   DATA[1675,3] := 1.0;
   DATA[1675,4] := 262.657;
   DATA[1675,5] := 8.46533;
   DATA[1675,6] := 319.4053;
   DATA[1675,8] := 1.0;
   DATA[1675,9] := 1.0;
   DATA[1675,10] := 1.0;
   DATA[1675,11] := 19.71957;
   DATA[1675,12] := 2.210037;
   DATA[1675,13] := 865.9639;
   DATA[1675,14] := 1.0;
   DATA[1675,15] := 2.0;
   DATA[1675,16] := 1.0;
   DATA[1675,17] := 1.0;
   DATA[1675,18] := 1.0;
   DATA[1675,19] := 2.0;
   DATA[1675,20] := 148.808;
   DATA[1675,21] := 153.9862;
   DATA[1675,22] := 1.713261;
   DATA[1675,23] := 801.756;
   DATA[1675,24] := 2.0;
   DATA[1675,25] := 2.0;
   DATA[1675,26] := 7.876058;
   DATA[1675,27] := 142.9377;
   DATA[1675,28] := 262.6891;
   DATA[1675,29] := 12.11228;
   DATA[1675,30] := 1.721866;
   DATA[1675,31] := 1.28372;
   DATA[1675,32] := 0.7355248;
   DATA[1675,33] := 0.3082983;
   DATA[1675,34] := 2.0;
   DATA[1675,35] := 249.7597;
   DATA[1675,36] := 1.585878;
   DATA[1675,37] := 188.7016;
   DATA[1675,38] := 0.000128152;
   DATA[1675,39] := 1.0;
   DATA[1676,1] := 815.3583;
   DATA[1676,2] := 1.0;
   DATA[1676,3] := 1.0;
   DATA[1676,4] := 262.657;
   DATA[1676,5] := 8.46533;
   DATA[1676,6] := 319.5334;
   DATA[1676,8] := 1.0;
   DATA[1676,9] := 1.0;
   DATA[1676,10] := 1.0;
   DATA[1676,11] := 19.71957;
   DATA[1676,12] := 2.210037;
   DATA[1676,13] := 865.323;
   DATA[1676,14] := 1.0;
   DATA[1676,15] := 2.0;
   DATA[1676,16] := 1.0;
   DATA[1676,17] := 1.0;
   DATA[1676,18] := 1.0;
   DATA[1676,19] := 2.0;
   DATA[1676,20] := 148.808;
   DATA[1676,21] := 153.9862;
   DATA[1676,22] := 1.713261;
   DATA[1676,23] := 801.756;
   DATA[1676,24] := 2.0;
   DATA[1676,25] := 2.0;
   DATA[1676,26] := 7.876058;
   DATA[1676,27] := 142.9633;
   DATA[1676,28] := 262.6891;
   DATA[1676,29] := 12.11228;
   DATA[1676,30] := 1.721866;
   DATA[1676,31] := 1.299731;
   DATA[1676,32] := 0.7355248;
   DATA[1676,33] := 0.3084265;
   DATA[1676,34] := 2.0;
   DATA[1676,35] := 249.7597;
   DATA[1676,36] := 1.585878;
   DATA[1676,37] := 188.7016;
   DATA[1676,38] := 0.000128152;
   DATA[1676,39] := 1.0;
   DATA[1677,1] := 815.5153;
   DATA[1677,2] := 1.0;
   DATA[1677,3] := 1.0;
   DATA[1677,4] := 262.657;
   DATA[1677,5] := 8.46533;
   DATA[1677,6] := 319.5334;
   DATA[1677,8] := 1.0;
   DATA[1677,9] := 1.0;
   DATA[1677,10] := 1.0;
   DATA[1677,11] := 19.70357;
   DATA[1677,12] := 2.210037;
   DATA[1677,13] := 865.0827;
   DATA[1677,14] := 1.0;
   DATA[1677,15] := 2.0;
   DATA[1677,16] := 1.0;
   DATA[1677,17] := 1.0;
   DATA[1677,18] := 1.0;
   DATA[1677,19] := 2.0;
   DATA[1677,20] := 148.808;
   DATA[1677,21] := 154.0631;
   DATA[1677,22] := 1.713261;
   DATA[1677,23] := 801.8329;
   DATA[1677,24] := 2.0;
   DATA[1677,25] := 2.0;
   DATA[1677,26] := 7.876058;
   DATA[1677,27] := 143.1172;
   DATA[1677,28] := 262.6891;
   DATA[1677,29] := 12.11228;
   DATA[1677,30] := 1.722892;
   DATA[1677,31] := 1.301652;
   DATA[1677,32] := 0.7355248;
   DATA[1677,33] := 0.3084905;
   DATA[1677,34] := 2.0;
   DATA[1677,35] := 249.8558;
   DATA[1677,36] := 1.585878;
   DATA[1677,37] := 188.7016;
   DATA[1677,38] := 0.000128152;
   DATA[1677,39] := 1.0;
   DATA[1678,1] := 815.5938;
   DATA[1678,2] := 1.0;
   DATA[1678,3] := 1.0;
   DATA[1678,4] := 262.657;
   DATA[1678,5] := 8.46533;
   DATA[1678,6] := 319.5334;
   DATA[1678,8] := 1.0;
   DATA[1678,9] := 1.0;
   DATA[1678,10] := 1.0;
   DATA[1678,11] := 19.68436;
   DATA[1678,12] := 2.210037;
   DATA[1678,13] := 864.4819;
   DATA[1678,14] := 1.0;
   DATA[1678,15] := 2.0;
   DATA[1678,16] := 1.0;
   DATA[1678,17] := 1.0;
   DATA[1678,18] := 1.0;
   DATA[1678,19] := 2.0;
   DATA[1678,20] := 148.808;
   DATA[1678,21] := 154.1912;
   DATA[1678,22] := 1.711082;
   DATA[1678,23] := 802.2174;
   DATA[1678,24] := 2.0;
   DATA[1678,25] := 2.0;
   DATA[1678,26] := 7.876058;
   DATA[1678,27] := 143.1172;
   DATA[1678,28] := 262.6891;
   DATA[1678,29] := 12.11228;
   DATA[1678,30] := 1.723789;
   DATA[1678,31] := 1.301652;
   DATA[1678,32] := 0.7355248;
   DATA[1678,33] := 0.3084905;
   DATA[1678,34] := 2.0;
   DATA[1678,35] := 249.9359;
   DATA[1678,36] := 1.585878;
   DATA[1678,37] := 188.7016;
   DATA[1678,38] := 0.000128152;
   DATA[1678,39] := 1.0;
   DATA[1679,1] := 815.4761;
   DATA[1679,2] := 1.0;
   DATA[1679,3] := 1.0;
   DATA[1679,4] := 262.657;
   DATA[1679,5] := 8.46533;
   DATA[1679,6] := 319.5334;
   DATA[1679,8] := 1.0;
   DATA[1679,9] := 1.0;
   DATA[1679,10] := 1.0;
   DATA[1679,11] := 19.68436;
   DATA[1679,12] := 2.210037;
   DATA[1679,13] := 864.2816;
   DATA[1679,14] := 1.0;
   DATA[1679,15] := 2.0;
   DATA[1679,16] := 1.0;
   DATA[1679,17] := 1.0;
   DATA[1679,18] := 1.0;
   DATA[1679,19] := 2.0;
   DATA[1679,20] := 148.808;
   DATA[1679,21] := 154.1912;
   DATA[1679,22] := 1.711082;
   DATA[1679,23] := 802.4097;
   DATA[1679,24] := 2.0;
   DATA[1679,25] := 2.0;
   DATA[1679,26] := 7.876058;
   DATA[1679,27] := 143.1172;
   DATA[1679,28] := 262.6891;
   DATA[1679,29] := 12.11228;
   DATA[1679,30] := 1.723789;
   DATA[1679,31] := 1.289484;
   DATA[1679,32] := 0.7355248;
   DATA[1679,33] := 0.3084905;
   DATA[1679,34] := 2.0;
   DATA[1679,35] := 249.9359;
   DATA[1679,36] := 1.585878;
   DATA[1679,37] := 188.7337;
   DATA[1679,38] := 0.000128152;
   DATA[1679,39] := 1.0;
   DATA[1680,1] := 815.3583;
   DATA[1680,2] := 1.0;
   DATA[1680,3] := 1.0;
   DATA[1680,4] := 262.657;
   DATA[1680,5] := 8.46533;
   DATA[1680,6] := 319.5334;
   DATA[1680,8] := 1.0;
   DATA[1680,9] := 1.0;
   DATA[1680,10] := 1.0;
   DATA[1680,11] := 19.68436;
   DATA[1680,12] := 2.210037;
   DATA[1680,13] := 863.7209;
   DATA[1680,14] := 1.0;
   DATA[1680,15] := 2.0;
   DATA[1680,16] := 1.0;
   DATA[1680,17] := 1.0;
   DATA[1680,18] := 1.0;
   DATA[1680,19] := 2.0;
   DATA[1680,20] := 148.808;
   DATA[1680,21] := 154.1912;
   DATA[1680,22] := 1.711082;
   DATA[1680,23] := 802.4866;
   DATA[1680,24] := 2.0;
   DATA[1680,25] := 2.0;
   DATA[1680,26] := 7.876058;
   DATA[1680,27] := 143.1172;
   DATA[1680,28] := 262.6891;
   DATA[1680,29] := 12.11228;
   DATA[1680,30] := 1.723789;
   DATA[1680,31] := 1.275522;
   DATA[1680,32] := 0.7355248;
   DATA[1680,33] := 0.3084905;
   DATA[1680,34] := 2.0;
   DATA[1680,35] := 249.9359;
   DATA[1680,36] := 1.601897;
   DATA[1680,37] := 188.8138;
   DATA[1680,38] := 0.000128152;
   DATA[1680,39] := 1.0;
   DATA[1681,1] := 815.319;
   DATA[1681,2] := 1.0;
   DATA[1681,3] := 1.0;
   DATA[1681,4] := 262.657;
   DATA[1681,5] := 8.46533;
   DATA[1681,6] := 319.5334;
   DATA[1681,8] := 1.0;
   DATA[1681,9] := 1.0;
   DATA[1681,10] := 1.0;
   DATA[1681,11] := 19.73238;
   DATA[1681,12] := 2.210037;
   DATA[1681,13] := 863.2402;
   DATA[1681,14] := 1.0;
   DATA[1681,15] := 2.0;
   DATA[1681,16] := 1.0;
   DATA[1681,17] := 1.0;
   DATA[1681,18] := 1.0;
   DATA[1681,19] := 2.0;
   DATA[1681,20] := 148.808;
   DATA[1681,21] := 154.1912;
   DATA[1681,22] := 1.711979;
   DATA[1681,23] := 802.871;
   DATA[1681,24] := 2.0;
   DATA[1681,25] := 2.0;
   DATA[1681,26] := 7.876058;
   DATA[1681,27] := 143.1172;
   DATA[1681,28] := 262.6891;
   DATA[1681,29] := 12.11228;
   DATA[1681,30] := 1.725327;
   DATA[1681,31] := 1.277315;
   DATA[1681,32] := 0.7355248;
   DATA[1681,33] := 0.3084905;
   DATA[1681,34] := 2.0;
   DATA[1681,35] := 249.9359;
   DATA[1681,36] := 1.681991;
   DATA[1681,37] := 188.8458;
   DATA[1681,38] := 0.000128152;
   DATA[1681,39] := 1.0;
   DATA[1682,1] := 815.319;
   DATA[1682,2] := 1.0;
   DATA[1682,3] := 1.0;
   DATA[1682,4] := 262.657;
   DATA[1682,5] := 8.46533;
   DATA[1682,6] := 319.5334;
   DATA[1682,8] := 1.0;
   DATA[1682,9] := 1.0;
   DATA[1682,10] := 1.0;
   DATA[1682,11] := 19.7868;
   DATA[1682,12] := 2.209397;
   DATA[1682,13] := 863.2803;
   DATA[1682,14] := 1.0;
   DATA[1682,15] := 2.0;
   DATA[1682,16] := 1.0;
   DATA[1682,17] := 1.0;
   DATA[1682,18] := 1.0;
   DATA[1682,19] := 2.0;
   DATA[1682,20] := 148.808;
   DATA[1682,21] := 154.1912;
   DATA[1682,22] := 1.712748;
   DATA[1682,23] := 803.4094;
   DATA[1682,24] := 2.0;
   DATA[1682,25] := 2.0;
   DATA[1682,26] := 7.876058;
   DATA[1682,27] := 143.0659;
   DATA[1682,28] := 262.6891;
   DATA[1682,29] := 12.11228;
   DATA[1682,30] := 1.725327;
   DATA[1682,31] := 1.276547;
   DATA[1682,32] := 0.7355248;
   DATA[1682,33] := 0.3084905;
   DATA[1682,34] := 2.0;
   DATA[1682,35] := 249.9359;
   DATA[1682,36] := 1.681991;
   DATA[1682,37] := 188.8458;
   DATA[1682,38] := 0.000128152;
   DATA[1682,39] := 1.0;
   DATA[1683,1] := 815.3975;
   DATA[1683,2] := 1.0;
   DATA[1683,3] := 1.0;
   DATA[1683,4] := 262.657;
   DATA[1683,5] := 8.46533;
   DATA[1683,6] := 319.5334;
   DATA[1683,8] := 1.0;
   DATA[1683,9] := 1.0;
   DATA[1683,10] := 1.0;
   DATA[1683,11] := 19.7868;
   DATA[1683,12] := 2.209397;
   DATA[1683,13] := 862.5593;
   DATA[1683,14] := 1.0;
   DATA[1683,15] := 2.0;
   DATA[1683,16] := 1.0;
   DATA[1683,17] := 1.0;
   DATA[1683,18] := 1.0;
   DATA[1683,19] := 2.0;
   DATA[1683,20] := 148.808;
   DATA[1683,21] := 154.1912;
   DATA[1683,22] := 1.712748;
   DATA[1683,23] := 803.4094;
   DATA[1683,24] := 2.0;
   DATA[1683,25] := 2.0;
   DATA[1683,26] := 7.876058;
   DATA[1683,27] := 143.0659;
   DATA[1683,28] := 262.6891;
   DATA[1683,29] := 12.11228;
   DATA[1683,30] := 1.725327;
   DATA[1683,31] := 1.27834;
   DATA[1683,32] := 0.7355248;
   DATA[1683,33] := 0.3084905;
   DATA[1683,34] := 2.0;
   DATA[1683,35] := 249.9359;
   DATA[1683,36] := 1.681991;
   DATA[1683,37] := 188.8458;
   DATA[1683,38] := 0.000128152;
   DATA[1683,39] := 1.0;
   DATA[1684,1] := 815.1228;
   DATA[1684,2] := 1.0;
   DATA[1684,3] := 1.0;
   DATA[1684,4] := 262.657;
   DATA[1684,5] := 8.46533;
   DATA[1684,6] := 319.5334;
   DATA[1684,8] := 1.0;
   DATA[1684,9] := 1.0;
   DATA[1684,10] := 1.0;
   DATA[1684,11] := 19.72277;
   DATA[1684,12] := 2.209397;
   DATA[1684,13] := 862.4391;
   DATA[1684,14] := 1.0;
   DATA[1684,15] := 2.0;
   DATA[1684,16] := 1.0;
   DATA[1684,17] := 1.0;
   DATA[1684,18] := 1.0;
   DATA[1684,19] := 2.0;
   DATA[1684,20] := 148.808;
   DATA[1684,21] := 154.1912;
   DATA[1684,22] := 1.712748;
   DATA[1684,23] := 803.8323;
   DATA[1684,24] := 2.0;
   DATA[1684,25] := 2.0;
   DATA[1684,26] := 7.876058;
   DATA[1684,27] := 143.0659;
   DATA[1684,28] := 262.6891;
   DATA[1684,29] := 12.11228;
   DATA[1684,30] := 1.725327;
   DATA[1684,31] := 1.272064;
   DATA[1684,32] := 0.7355248;
   DATA[1684,33] := 0.3084905;
   DATA[1684,34] := 2.0;
   DATA[1684,35] := 249.9359;
   DATA[1684,36] := 1.665972;
   DATA[1684,37] := 188.8458;
   DATA[1684,38] := 0.000128152;
   DATA[1684,39] := 1.0;
   DATA[1685,1] := 815.0835;
   DATA[1685,2] := 1.0;
   DATA[1685,3] := 1.0;
   DATA[1685,4] := 262.657;
   DATA[1685,5] := 8.46533;
   DATA[1685,6] := 319.5334;
   DATA[1685,8] := 1.0;
   DATA[1685,9] := 1.0;
   DATA[1685,10] := 1.0;
   DATA[1685,11] := 19.70357;
   DATA[1685,12] := 2.209397;
   DATA[1685,13] := 862.0386;
   DATA[1685,14] := 1.0;
   DATA[1685,15] := 2.0;
   DATA[1685,16] := 1.0;
   DATA[1685,17] := 1.0;
   DATA[1685,18] := 1.0;
   DATA[1685,19] := 2.0;
   DATA[1685,20] := 148.808;
   DATA[1685,21] := 154.1912;
   DATA[1685,22] := 1.712876;
   DATA[1685,23] := 803.6016;
   DATA[1685,24] := 2.0;
   DATA[1685,25] := 2.0;
   DATA[1685,26] := 7.876058;
   DATA[1685,27] := 143.0659;
   DATA[1685,28] := 262.6891;
   DATA[1685,29] := 12.11228;
   DATA[1685,30] := 1.725327;
   DATA[1685,31] := 1.271935;
   DATA[1685,32] := 0.7355248;
   DATA[1685,33] := 0.3084905;
   DATA[1685,34] := 2.0;
   DATA[1685,35] := 249.9359;
   DATA[1685,36] := 1.649953;
   DATA[1685,37] := 188.8458;
   DATA[1685,38] := 0.000128152;
   DATA[1685,39] := 1.0;
   DATA[1686,1] := 815.3975;
   DATA[1686,2] := 1.0;
   DATA[1686,3] := 1.0;
   DATA[1686,4] := 262.657;
   DATA[1686,5] := 8.46533;
   DATA[1686,6] := 319.5334;
   DATA[1686,8] := 1.0;
   DATA[1686,9] := 1.0;
   DATA[1686,10] := 1.0;
   DATA[1686,11] := 19.70357;
   DATA[1686,12] := 2.209397;
   DATA[1686,13] := 861.7582;
   DATA[1686,14] := 1.0;
   DATA[1686,15] := 2.0;
   DATA[1686,16] := 1.0;
   DATA[1686,17] := 1.0;
   DATA[1686,18] := 1.0;
   DATA[1686,19] := 2.0;
   DATA[1686,20] := 148.808;
   DATA[1686,21] := 154.1912;
   DATA[1686,22] := 1.712876;
   DATA[1686,23] := 803.6016;
   DATA[1686,24] := 2.0;
   DATA[1686,25] := 2.0;
   DATA[1686,26] := 7.876058;
   DATA[1686,27] := 143.0659;
   DATA[1686,28] := 262.6891;
   DATA[1686,29] := 12.11228;
   DATA[1686,30] := 1.725327;
   DATA[1686,31] := 1.270911;
   DATA[1686,32] := 0.7355248;
   DATA[1686,33] := 0.3084905;
   DATA[1686,34] := 2.0;
   DATA[1686,35] := 249.9359;
   DATA[1686,36] := 1.649953;
   DATA[1686,37] := 188.8458;
   DATA[1686,38] := 0.000128152;
   DATA[1686,39] := 1.0;
   DATA[1687,1] := 815.2798;
   DATA[1687,2] := 1.0;
   DATA[1687,3] := 1.0;
   DATA[1687,4] := 262.657;
   DATA[1687,5] := 8.46533;
   DATA[1687,6] := 319.5334;
   DATA[1687,8] := 1.0;
   DATA[1687,9] := 1.0;
   DATA[1687,10] := 1.0;
   DATA[1687,11] := 19.76439;
   DATA[1687,12] := 2.214649;
   DATA[1687,13] := 860.9572;
   DATA[1687,14] := 1.0;
   DATA[1687,15] := 2.0;
   DATA[1687,16] := 1.0;
   DATA[1687,17] := 1.0;
   DATA[1687,18] := 1.0;
   DATA[1687,19] := 2.0;
   DATA[1687,20] := 148.808;
   DATA[1687,21] := 154.1912;
   DATA[1687,22] := 1.712876;
   DATA[1687,23] := 803.4094;
   DATA[1687,24] := 2.0;
   DATA[1687,25] := 2.0;
   DATA[1687,26] := 7.876058;
   DATA[1687,27] := 143.0659;
   DATA[1687,28] := 262.6891;
   DATA[1687,29] := 12.11228;
   DATA[1687,30] := 1.724045;
   DATA[1687,31] := 1.270398;
   DATA[1687,32] := 0.7355248;
   DATA[1687,33] := 0.3084905;
   DATA[1687,34] := 2.0;
   DATA[1687,35] := 249.9359;
   DATA[1687,36] := 1.649953;
   DATA[1687,37] := 188.8458;
   DATA[1687,38] := 0.000128152;
   DATA[1687,39] := 1.0;
   DATA[1688,1] := 815.2013;
   DATA[1688,2] := 1.0;
   DATA[1688,3] := 1.0;
   DATA[1688,4] := 262.657;
   DATA[1688,5] := 8.46533;
   DATA[1688,6] := 319.5334;
   DATA[1688,8] := 1.0;
   DATA[1688,9] := 1.0;
   DATA[1688,10] := 1.0;
   DATA[1688,11] := 19.76439;
   DATA[1688,12] := 2.214649;
   DATA[1688,13] := 860.5566;
   DATA[1688,14] := 1.0;
   DATA[1688,15] := 2.0;
   DATA[1688,16] := 1.0;
   DATA[1688,17] := 1.0;
   DATA[1688,18] := 1.0;
   DATA[1688,19] := 2.0;
   DATA[1688,20] := 148.808;
   DATA[1688,21] := 154.1912;
   DATA[1688,22] := 1.712876;
   DATA[1688,23] := 803.294;
   DATA[1688,24] := 2.0;
   DATA[1688,25] := 2.0;
   DATA[1688,26] := 7.876058;
   DATA[1688,27] := 143.0659;
   DATA[1688,28] := 262.6891;
   DATA[1688,29] := 12.11228;
   DATA[1688,30] := 1.724045;
   DATA[1688,31] := 1.287306;
   DATA[1688,32] := 0.7355248;
   DATA[1688,33] := 0.3084905;
   DATA[1688,34] := 2.0;
   DATA[1688,35] := 249.9359;
   DATA[1688,36] := 1.649953;
   DATA[1688,37] := 188.8458;
   DATA[1688,38] := 0.000128152;
   DATA[1688,39] := 1.0;
   DATA[1689,1] := 815.4761;
   DATA[1689,2] := 1.0;
   DATA[1689,3] := 1.0;
   DATA[1689,4] := 262.657;
   DATA[1689,5] := 8.46533;
   DATA[1689,6] := 319.5334;
   DATA[1689,8] := 1.0;
   DATA[1689,9] := 1.0;
   DATA[1689,10] := 1.0;
   DATA[1689,11] := 19.77399;
   DATA[1689,12] := 2.215418;
   DATA[1689,13] := 860.0359;
   DATA[1689,14] := 1.0;
   DATA[1689,15] := 2.0;
   DATA[1689,16] := 1.0;
   DATA[1689,17] := 1.0;
   DATA[1689,18] := 1.0;
   DATA[1689,19] := 2.0;
   DATA[1689,20] := 148.808;
   DATA[1689,21] := 154.1912;
   DATA[1689,22] := 1.712876;
   DATA[1689,23] := 803.4863;
   DATA[1689,24] := 2.0;
   DATA[1689,25] := 2.0;
   DATA[1689,26] := 7.876058;
   DATA[1689,27] := 143.0659;
   DATA[1689,28] := 262.6891;
   DATA[1689,29] := 12.11228;
   DATA[1689,30] := 1.722251;
   DATA[1689,31] := 1.291918;
   DATA[1689,32] := 0.7355248;
   DATA[1689,33] := 0.3084905;
   DATA[1689,34] := 2.0;
   DATA[1689,35] := 249.9359;
   DATA[1689,36] := 1.649953;
   DATA[1689,37] := 188.8458;
   DATA[1689,38] := 0.000128152;
   DATA[1689,39] := 1.0;
   DATA[1690,1] := 815.2013;
   DATA[1690,2] := 1.0;
   DATA[1690,3] := 1.0;
   DATA[1690,4] := 262.657;
   DATA[1690,5] := 8.46533;
   DATA[1690,6] := 319.5334;
   DATA[1690,8] := 1.0;
   DATA[1690,9] := 1.0;
   DATA[1690,10] := 1.0;
   DATA[1690,11] := 19.7804;
   DATA[1690,12] := 2.21593;
   DATA[1690,13] := 859.8757;
   DATA[1690,14] := 1.0;
   DATA[1690,15] := 2.0;
   DATA[1690,16] := 1.0;
   DATA[1690,17] := 1.0;
   DATA[1690,18] := 1.0;
   DATA[1690,19] := 2.0;
   DATA[1690,20] := 148.808;
   DATA[1690,21] := 154.1912;
   DATA[1690,22] := 1.712876;
   DATA[1690,23] := 803.6401;
   DATA[1690,24] := 2.0;
   DATA[1690,25] := 2.0;
   DATA[1690,26] := 7.876058;
   DATA[1690,27] := 143.0659;
   DATA[1690,28] := 262.6891;
   DATA[1690,29] := 12.11228;
   DATA[1690,30] := 1.721866;
   DATA[1690,31] := 1.291918;
   DATA[1690,32] := 0.7355248;
   DATA[1690,33] := 0.3084905;
   DATA[1690,34] := 2.0;
   DATA[1690,35] := 250.0961;
   DATA[1690,36] := 1.649953;
   DATA[1690,37] := 188.8458;
   DATA[1690,38] := 0.000128152;
   DATA[1690,39] := 1.0;
   DATA[1691,1] := 815.0835;
   DATA[1691,2] := 1.0;
   DATA[1691,3] := 1.0;
   DATA[1691,4] := 262.657;
   DATA[1691,5] := 8.46533;
   DATA[1691,6] := 319.5334;
   DATA[1691,8] := 1.0;
   DATA[1691,9] := 1.0;
   DATA[1691,10] := 1.0;
   DATA[1691,11] := 19.7804;
   DATA[1691,12] := 2.21593;
   DATA[1691,13] := 858.8743;
   DATA[1691,14] := 1.0;
   DATA[1691,15] := 2.0;
   DATA[1691,16] := 1.0;
   DATA[1691,17] := 1.0;
   DATA[1691,18] := 1.0;
   DATA[1691,19] := 2.0;
   DATA[1691,20] := 148.808;
   DATA[1691,21] := 154.1912;
   DATA[1691,22] := 1.712107;
   DATA[1691,23] := 803.8323;
   DATA[1691,24] := 2.0;
   DATA[1691,25] := 2.0;
   DATA[1691,26] := 7.876058;
   DATA[1691,27] := 143.0659;
   DATA[1691,28] := 262.6891;
   DATA[1691,29] := 12.11228;
   DATA[1691,30] := 1.721866;
   DATA[1691,31] := 1.282567;
   DATA[1691,32] := 0.7355248;
   DATA[1691,33] := 0.3084905;
   DATA[1691,34] := 2.0;
   DATA[1691,35] := 250.0961;
   DATA[1691,36] := 1.537821;
   DATA[1691,37] := 188.8458;
   DATA[1691,38] := 0.000128152;
   DATA[1691,39] := 1.0;
   DATA[1692,1] := 814.8088;
   DATA[1692,2] := 1.0;
   DATA[1692,3] := 1.0;
   DATA[1692,4] := 262.657;
   DATA[1692,5] := 8.46533;
   DATA[1692,6] := 319.5334;
   DATA[1692,8] := 1.0;
   DATA[1692,9] := 1.0;
   DATA[1692,10] := 1.0;
   DATA[1692,11] := 19.80601;
   DATA[1692,12] := 2.21593;
   DATA[1692,13] := 858.3536;
   DATA[1692,14] := 1.0;
   DATA[1692,15] := 2.0;
   DATA[1692,16] := 1.0;
   DATA[1692,17] := 1.0;
   DATA[1692,18] := 1.0;
   DATA[1692,19] := 2.0;
   DATA[1692,20] := 148.808;
   DATA[1692,21] := 154.1912;
   DATA[1692,22] := 1.710057;
   DATA[1692,23] := 804.4476;
   DATA[1692,24] := 2.0;
   DATA[1692,25] := 2.0;
   DATA[1692,26] := 7.876058;
   DATA[1692,27] := 143.0659;
   DATA[1692,28] := 262.6891;
   DATA[1692,29] := 12.11228;
   DATA[1692,30] := 1.721866;
   DATA[1692,31] := 1.281927;
   DATA[1692,32] := 0.7353967;
   DATA[1692,33] := 0.3084905;
   DATA[1692,34] := 2.0;
   DATA[1692,35] := 250.0961;
   DATA[1692,36] := 1.537821;
   DATA[1692,37] := 188.8458;
   DATA[1692,38] := 0.000128152;
   DATA[1692,39] := 1.0;
   DATA[1693,1] := 814.7302;
   DATA[1693,2] := 1.0;
   DATA[1693,3] := 1.0;
   DATA[1693,4] := 262.657;
   DATA[1693,5] := 8.46533;
   DATA[1693,6] := 319.5334;
   DATA[1693,8] := 1.0;
   DATA[1693,9] := 1.0;
   DATA[1693,10] := 1.0;
   DATA[1693,11] := 19.83802;
   DATA[1693,12] := 2.21593;
   DATA[1693,13] := 857.6327;
   DATA[1693,14] := 1.0;
   DATA[1693,15] := 2.0;
   DATA[1693,16] := 1.0;
   DATA[1693,17] := 1.0;
   DATA[1693,18] := 1.0;
   DATA[1693,19] := 2.0;
   DATA[1693,20] := 148.808;
   DATA[1693,21] := 154.1912;
   DATA[1693,22] := 1.710057;
   DATA[1693,23] := 804.7167;
   DATA[1693,24] := 2.0;
   DATA[1693,25] := 2.0;
   DATA[1693,26] := 7.876058;
   DATA[1693,27] := 143.0659;
   DATA[1693,28] := 262.6891;
   DATA[1693,29] := 12.11228;
   DATA[1693,30] := 1.721866;
   DATA[1693,31] := 1.281927;
   DATA[1693,32] := 0.7353967;
   DATA[1693,33] := 0.3084905;
   DATA[1693,34] := 2.0;
   DATA[1693,35] := 250.016;
   DATA[1693,36] := 1.569859;
   DATA[1693,37] := 188.8458;
   DATA[1693,38] := 0.000128152;
   DATA[1693,39] := 1.0;
   DATA[1694,1] := 814.7302;
   DATA[1694,2] := 1.0;
   DATA[1694,3] := 1.0;
   DATA[1694,4] := 262.657;
   DATA[1694,5] := 8.46533;
   DATA[1694,6] := 319.5334;
   DATA[1694,8] := 1.0;
   DATA[1694,9] := 1.0;
   DATA[1694,10] := 1.0;
   DATA[1694,11] := 19.83802;
   DATA[1694,12] := 2.21593;
   DATA[1694,13] := 857.6327;
   DATA[1694,14] := 1.0;
   DATA[1694,15] := 2.0;
   DATA[1694,16] := 1.0;
   DATA[1694,17] := 1.0;
   DATA[1694,18] := 1.0;
   DATA[1694,19] := 2.0;
   DATA[1694,20] := 148.808;
   DATA[1694,21] := 154.1912;
   DATA[1694,22] := 1.710057;
   DATA[1694,23] := 804.7167;
   DATA[1694,24] := 2.0;
   DATA[1694,25] := 2.0;
   DATA[1694,26] := 7.876058;
   DATA[1694,27] := 143.0659;
   DATA[1694,28] := 262.6891;
   DATA[1694,29] := 12.11228;
   DATA[1694,30] := 1.721866;
   DATA[1694,31] := 1.281927;
   DATA[1694,32] := 0.7353967;
   DATA[1694,33] := 0.3084905;
   DATA[1694,34] := 2.0;
   DATA[1694,35] := 250.016;
   DATA[1694,36] := 1.569859;
   DATA[1694,37] := 188.8458;
   DATA[1694,38] := 0.000128152;
   DATA[1694,39] := 1.0;
   DATA[1695,1] := 814.8088;
   DATA[1695,2] := 1.0;
   DATA[1695,3] := 1.0;
   DATA[1695,4] := 262.657;
   DATA[1695,5] := 8.46533;
   DATA[1695,6] := 319.5334;
   DATA[1695,8] := 1.0;
   DATA[1695,9] := 1.0;
   DATA[1695,10] := 1.0;
   DATA[1695,11] := 19.83802;
   DATA[1695,12] := 2.21593;
   DATA[1695,13] := 857.3523;
   DATA[1695,14] := 1.0;
   DATA[1695,15] := 2.0;
   DATA[1695,16] := 1.0;
   DATA[1695,17] := 1.0;
   DATA[1695,18] := 1.0;
   DATA[1695,19] := 2.0;
   DATA[1695,20] := 148.808;
   DATA[1695,21] := 154.1912;
   DATA[1695,22] := 1.710057;
   DATA[1695,23] := 804.6398;
   DATA[1695,24] := 2.0;
   DATA[1695,25] := 2.0;
   DATA[1695,26] := 7.876058;
   DATA[1695,27] := 143.2197;
   DATA[1695,28] := 262.6891;
   DATA[1695,29] := 12.11228;
   DATA[1695,30] := 1.721866;
   DATA[1695,31] := 1.290509;
   DATA[1695,32] := 0.7353967;
   DATA[1695,33] := 0.3084905;
   DATA[1695,34] := 2.0;
   DATA[1695,35] := 249.984;
   DATA[1695,36] := 1.681991;
   DATA[1695,37] := 188.8458;
   DATA[1695,38] := 0.000128152;
   DATA[1695,39] := 1.0;
   DATA[1696,1] := 814.9265;
   DATA[1696,2] := 1.0;
   DATA[1696,3] := 1.0;
   DATA[1696,4] := 262.657;
   DATA[1696,5] := 8.46533;
   DATA[1696,6] := 319.5334;
   DATA[1696,8] := 1.0;
   DATA[1696,9] := 1.0;
   DATA[1696,10] := 1.0;
   DATA[1696,11] := 19.83802;
   DATA[1696,12] := 2.21593;
   DATA[1696,13] := 856.8716;
   DATA[1696,14] := 1.0;
   DATA[1696,15] := 2.0;
   DATA[1696,16] := 1.0;
   DATA[1696,17] := 1.0;
   DATA[1696,18] := 1.0;
   DATA[1696,19] := 2.0;
   DATA[1696,20] := 148.808;
   DATA[1696,21] := 154.1912;
   DATA[1696,22] := 1.711595;
   DATA[1696,23] := 804.3707;
   DATA[1696,24] := 2.0;
   DATA[1696,25] := 2.0;
   DATA[1696,26] := 7.876058;
   DATA[1696,27] := 143.2197;
   DATA[1696,28] := 262.6891;
   DATA[1696,29] := 12.11228;
   DATA[1696,30] := 1.722892;
   DATA[1696,31] := 1.291789;
   DATA[1696,32] := 0.7353967;
   DATA[1696,33] := 0.3084905;
   DATA[1696,34] := 2.0;
   DATA[1696,35] := 249.984;
   DATA[1696,36] := 1.681991;
   DATA[1696,37] := 188.8458;
   DATA[1696,38] := 0.000128152;
   DATA[1696,39] := 1.0;
   DATA[1697,1] := 814.8088;
   DATA[1697,2] := 1.0;
   DATA[1697,3] := 1.0;
   DATA[1697,4] := 262.657;
   DATA[1697,5] := 8.46533;
   DATA[1697,6] := 319.5334;
   DATA[1697,8] := 1.0;
   DATA[1697,9] := 1.0;
   DATA[1697,10] := 1.0;
   DATA[1697,11] := 19.73878;
   DATA[1697,12] := 2.214265;
   DATA[1697,13] := 856.9117;
   DATA[1697,14] := 1.0;
   DATA[1697,15] := 2.0;
   DATA[1697,16] := 1.0;
   DATA[1697,17] := 1.0;
   DATA[1697,18] := 1.0;
   DATA[1697,19] := 2.0;
   DATA[1697,20] := 148.808;
   DATA[1697,21] := 154.1912;
   DATA[1697,22] := 1.711595;
   DATA[1697,23] := 804.0246;
   DATA[1697,24] := 2.0;
   DATA[1697,25] := 2.0;
   DATA[1697,26] := 7.876058;
   DATA[1697,27] := 143.2197;
   DATA[1697,28] := 262.625;
   DATA[1697,29] := 12.11228;
   DATA[1697,30] := 1.723661;
   DATA[1697,31] := 1.282439;
   DATA[1697,32] := 0.7353967;
   DATA[1697,33] := 0.3084905;
   DATA[1697,34] := 2.0;
   DATA[1697,35] := 249.984;
   DATA[1697,36] := 1.681991;
   DATA[1697,37] := 188.8458;
   DATA[1697,38] := 0.000128152;
   DATA[1697,39] := 1.0;
   DATA[1698,1] := 815.162;
   DATA[1698,2] := 1.0;
   DATA[1698,3] := 1.0;
   DATA[1698,4] := 262.657;
   DATA[1698,5] := 8.46533;
   DATA[1698,6] := 319.5334;
   DATA[1698,8] := 1.0;
   DATA[1698,9] := 1.0;
   DATA[1698,10] := 1.0;
   DATA[1698,11] := 19.70357;
   DATA[1698,12] := 2.214265;
   DATA[1698,13] := 856.0706;
   DATA[1698,14] := 1.0;
   DATA[1698,15] := 2.0;
   DATA[1698,16] := 1.0;
   DATA[1698,17] := 1.0;
   DATA[1698,18] := 1.0;
   DATA[1698,19] := 2.0;
   DATA[1698,20] := 148.808;
   DATA[1698,21] := 154.1912;
   DATA[1698,22] := 1.711595;
   DATA[1698,23] := 804.8321;
   DATA[1698,24] := 2.0;
   DATA[1698,25] := 2.0;
   DATA[1698,26] := 7.876058;
   DATA[1698,27] := 143.2197;
   DATA[1698,28] := 262.3366;
   DATA[1698,29] := 12.11228;
   DATA[1698,30] := 1.723661;
   DATA[1698,31] := 1.282439;
   DATA[1698,32] := 0.7353967;
   DATA[1698,33] := 0.3084905;
   DATA[1698,34] := 2.0;
   DATA[1698,35] := 249.984;
   DATA[1698,36] := 1.681991;
   DATA[1698,37] := 188.8458;
   DATA[1698,38] := 0.000128152;
   DATA[1698,39] := 1.0;
   DATA[1699,1] := 815.0835;
   DATA[1699,2] := 1.0;
   DATA[1699,3] := 1.0;
   DATA[1699,4] := 262.657;
   DATA[1699,5] := 8.46533;
   DATA[1699,6] := 319.5334;
   DATA[1699,8] := 1.0;
   DATA[1699,9] := 1.0;
   DATA[1699,10] := 1.0;
   DATA[1699,11] := 19.70357;
   DATA[1699,12] := 2.214265;
   DATA[1699,13] := 855.8303;
   DATA[1699,14] := 1.0;
   DATA[1699,15] := 2.0;
   DATA[1699,16] := 1.0;
   DATA[1699,17] := 1.0;
   DATA[1699,18] := 1.0;
   DATA[1699,19] := 2.0;
   DATA[1699,20] := 148.808;
   DATA[1699,21] := 154.1912;
   DATA[1699,22] := 1.711595;
   DATA[1699,23] := 804.4476;
   DATA[1699,24] := 2.0;
   DATA[1699,25] := 2.0;
   DATA[1699,26] := 7.876058;
   DATA[1699,27] := 143.2197;
   DATA[1699,28] := 262.3366;
   DATA[1699,29] := 12.11228;
   DATA[1699,30] := 1.723661;
   DATA[1699,31] := 1.282439;
   DATA[1699,32] := 0.7353967;
   DATA[1699,33] := 0.3084905;
   DATA[1699,34] := 2.0;
   DATA[1699,35] := 249.984;
   DATA[1699,36] := 1.681991;
   DATA[1699,37] := 188.8458;
   DATA[1699,38] := 0.000128152;
   DATA[1699,39] := 1.0;
   DATA[1700,1] := 814.8873;
   DATA[1700,2] := 1.0;
   DATA[1700,3] := 1.0;
   DATA[1700,4] := 262.625;
   DATA[1700,5] := 8.46533;
   DATA[1700,6] := 319.5334;
   DATA[1700,8] := 1.0;
   DATA[1700,9] := 1.0;
   DATA[1700,10] := 1.0;
   DATA[1700,11] := 19.70357;
   DATA[1700,12] := 2.214265;
   DATA[1700,13] := 854.9491;
   DATA[1700,14] := 1.0;
   DATA[1700,15] := 2.0;
   DATA[1700,16] := 1.0;
   DATA[1700,17] := 1.0;
   DATA[1700,18] := 1.0;
   DATA[1700,19] := 2.0;
   DATA[1700,20] := 148.808;
   DATA[1700,21] := 154.1912;
   DATA[1700,22] := 1.711595;
   DATA[1700,23] := 804.6014;
   DATA[1700,24] := 2.0;
   DATA[1700,25] := 2.0;
   DATA[1700,26] := 7.876058;
   DATA[1700,27] := 143.2197;
   DATA[1700,28] := 262.3366;
   DATA[1700,29] := 12.11228;
   DATA[1700,30] := 1.723661;
   DATA[1700,31] := 1.282439;
   DATA[1700,32] := 0.7353967;
   DATA[1700,33] := 0.3084905;
   DATA[1700,34] := 2.0;
   DATA[1700,35] := 249.984;
   DATA[1700,36] := 1.681991;
   DATA[1700,37] := 188.8458;
   DATA[1700,38] := 0.000128152;
   DATA[1700,39] := 1.0;
   DATA[1701,1] := 815.1228;
   DATA[1701,2] := 1.0;
   DATA[1701,3] := 1.0;
   DATA[1701,4] := 262.625;
   DATA[1701,5] := 8.46533;
   DATA[1701,6] := 319.5334;
   DATA[1701,8] := 1.0;
   DATA[1701,9] := 1.0;
   DATA[1701,10] := 1.0;
   DATA[1701,11] := 19.75799;
   DATA[1701,12] := 2.212728;
   DATA[1701,13] := 854.7087;
   DATA[1701,14] := 1.0;
   DATA[1701,15] := 2.0;
   DATA[1701,16] := 1.0;
   DATA[1701,17] := 1.0;
   DATA[1701,18] := 1.0;
   DATA[1701,19] := 2.0;
   DATA[1701,20] := 148.808;
   DATA[1701,21] := 154.1912;
   DATA[1701,22] := 1.711595;
   DATA[1701,23] := 804.909;
   DATA[1701,24] := 2.0;
   DATA[1701,25] := 2.0;
   DATA[1701,26] := 7.876058;
   DATA[1701,27] := 143.2197;
   DATA[1701,28] := 262.3366;
   DATA[1701,29] := 12.11228;
   DATA[1701,30] := 1.723661;
   DATA[1701,31] := 1.274241;
   DATA[1701,32] := 0.7353967;
   DATA[1701,33] := 0.3084905;
   DATA[1701,34] := 2.0;
   DATA[1701,35] := 249.984;
   DATA[1701,36] := 1.681991;
   DATA[1701,37] := 188.8458;
   DATA[1701,38] := 0.000128152;
   DATA[1701,39] := 1.0;
   DATA[1702,1] := 815.3583;
   DATA[1702,2] := 1.0;
   DATA[1702,3] := 1.0;
   DATA[1702,4] := 262.625;
   DATA[1702,5] := 8.46533;
   DATA[1702,6] := 319.5334;
   DATA[1702,8] := 1.0;
   DATA[1702,9] := 1.0;
   DATA[1702,10] := 1.0;
   DATA[1702,11] := 19.75799;
   DATA[1702,12] := 2.211959;
   DATA[1702,13] := 854.0679;
   DATA[1702,14] := 1.0;
   DATA[1702,15] := 2.0;
   DATA[1702,16] := 1.0;
   DATA[1702,17] := 1.0;
   DATA[1702,18] := 1.0;
   DATA[1702,19] := 2.0;
   DATA[1702,20] := 148.808;
   DATA[1702,21] := 154.1912;
   DATA[1702,22] := 1.711595;
   DATA[1702,23] := 804.7552;
   DATA[1702,24] := 2.0;
   DATA[1702,25] := 2.0;
   DATA[1702,26] := 7.876058;
   DATA[1702,27] := 143.2197;
   DATA[1702,28] := 262.657;
   DATA[1702,29] := 12.11228;
   DATA[1702,30] := 1.723661;
   DATA[1702,31] := 1.26361;
   DATA[1702,32] := 0.7353967;
   DATA[1702,33] := 0.3084905;
   DATA[1702,34] := 2.0;
   DATA[1702,35] := 249.984;
   DATA[1702,36] := 1.681991;
   DATA[1702,37] := 188.8458;
   DATA[1702,38] := 0.000128152;
   DATA[1702,39] := 1.0;
   DATA[1703,1] := 815.2798;
   DATA[1703,2] := 1.0;
   DATA[1703,3] := 1.0;
   DATA[1703,4] := 262.625;
   DATA[1703,5] := 8.46533;
   DATA[1703,6] := 319.5334;
   DATA[1703,8] := 1.0;
   DATA[1703,9] := 1.0;
   DATA[1703,10] := 1.0;
   DATA[1703,11] := 19.75799;
   DATA[1703,12] := 2.211959;
   DATA[1703,13] := 853.3469;
   DATA[1703,14] := 1.0;
   DATA[1703,15] := 2.0;
   DATA[1703,16] := 1.0;
   DATA[1703,17] := 1.0;
   DATA[1703,18] := 1.0;
   DATA[1703,19] := 2.0;
   DATA[1703,20] := 148.808;
   DATA[1703,21] := 154.1912;
   DATA[1703,22] := 1.711595;
   DATA[1703,23] := 804.6398;
   DATA[1703,24] := 2.0;
   DATA[1703,25] := 2.0;
   DATA[1703,26] := 7.876058;
   DATA[1703,27] := 143.2197;
   DATA[1703,28] := 262.657;
   DATA[1703,29] := 12.11228;
   DATA[1703,30] := 1.723661;
   DATA[1703,31] := 1.260792;
   DATA[1703,32] := 0.7353967;
   DATA[1703,33] := 0.3084905;
   DATA[1703,34] := 2.0;
   DATA[1703,35] := 249.984;
   DATA[1703,36] := 1.681991;
   DATA[1703,37] := 188.8458;
   DATA[1703,38] := 0.000128152;
   DATA[1703,39] := 1.0;
   DATA[1704,1] := 815.319;
   DATA[1704,2] := 1.0;
   DATA[1704,3] := 1.0;
   DATA[1704,4] := 262.625;
   DATA[1704,5] := 8.46533;
   DATA[1704,6] := 319.5334;
   DATA[1704,8] := 1.0;
   DATA[1704,9] := 1.0;
   DATA[1704,10] := 1.0;
   DATA[1704,11] := 19.74198;
   DATA[1704,12] := 2.211959;
   DATA[1704,13] := 853.3469;
   DATA[1704,14] := 1.0;
   DATA[1704,15] := 2.0;
   DATA[1704,16] := 1.0;
   DATA[1704,17] := 1.0;
   DATA[1704,18] := 1.0;
   DATA[1704,19] := 2.0;
   DATA[1704,20] := 148.808;
   DATA[1704,21] := 154.1912;
   DATA[1704,22] := 1.711595;
   DATA[1704,23] := 804.6398;
   DATA[1704,24] := 2.0;
   DATA[1704,25] := 2.0;
   DATA[1704,26] := 7.876058;
   DATA[1704,27] := 143.2197;
   DATA[1704,28] := 262.657;
   DATA[1704,29] := 12.11228;
   DATA[1704,30] := 1.723661;
   DATA[1704,31] := 1.260792;
   DATA[1704,32] := 0.7353967;
   DATA[1704,33] := 0.3084905;
   DATA[1704,34] := 2.0;
   DATA[1704,35] := 249.984;
   DATA[1704,36] := 1.681991;
   DATA[1704,37] := 188.8458;
   DATA[1704,38] := 0.000128152;
   DATA[1704,39] := 1.0;
   DATA[1705,1] := 815.162;
   DATA[1705,2] := 1.0;
   DATA[1705,3] := 1.0;
   DATA[1705,4] := 262.625;
   DATA[1705,5] := 8.46533;
   DATA[1705,6] := 319.5334;
   DATA[1705,8] := 1.0;
   DATA[1705,9] := 1.0;
   DATA[1705,10] := 1.0;
   DATA[1705,11] := 19.73878;
   DATA[1705,12] := 2.209653;
   DATA[1705,13] := 852.666;
   DATA[1705,14] := 1.0;
   DATA[1705,15] := 2.0;
   DATA[1705,16] := 1.0;
   DATA[1705,17] := 1.0;
   DATA[1705,18] := 1.0;
   DATA[1705,19] := 2.0;
   DATA[1705,20] := 148.808;
   DATA[1705,21] := 154.1912;
   DATA[1705,22] := 1.711595;
   DATA[1705,23] := 804.909;
   DATA[1705,24] := 2.0;
   DATA[1705,25] := 2.0;
   DATA[1705,26] := 7.876058;
   DATA[1705,27] := 143.2197;
   DATA[1705,28] := 262.657;
   DATA[1705,29] := 12.11228;
   DATA[1705,30] := 1.723661;
   DATA[1705,31] := 1.265787;
   DATA[1705,32] := 0.7353967;
   DATA[1705,33] := 0.3084905;
   DATA[1705,34] := 2.0;
   DATA[1705,35] := 249.984;
   DATA[1705,36] := 1.681991;
   DATA[1705,37] := 188.8458;
   DATA[1705,38] := 0.000128152;
   DATA[1705,39] := 1.0;
   DATA[1706,1] := 815.2798;
   DATA[1706,2] := 1.0;
   DATA[1706,3] := 1.0;
   DATA[1706,4] := 262.625;
   DATA[1706,5] := 8.46533;
   DATA[1706,6] := 319.5334;
   DATA[1706,8] := 1.0;
   DATA[1706,9] := 1.0;
   DATA[1706,10] := 1.0;
   DATA[1706,11] := 19.73878;
   DATA[1706,12] := 2.209653;
   DATA[1706,13] := 852.1453;
   DATA[1706,14] := 1.0;
   DATA[1706,15] := 2.0;
   DATA[1706,16] := 1.0;
   DATA[1706,17] := 1.0;
   DATA[1706,18] := 1.0;
   DATA[1706,19] := 2.0;
   DATA[1706,20] := 148.808;
   DATA[1706,21] := 154.1912;
   DATA[1706,22] := 1.710826;
   DATA[1706,23] := 804.7936;
   DATA[1706,24] := 2.0;
   DATA[1706,25] := 2.0;
   DATA[1706,26] := 7.876058;
   DATA[1706,27] := 143.2197;
   DATA[1706,28] := 262.657;
   DATA[1706,29] := 12.11228;
   DATA[1706,30] := 1.723661;
   DATA[1706,31] := 1.271039;
   DATA[1706,32] := 0.7353967;
   DATA[1706,33] := 0.3084905;
   DATA[1706,34] := 2.0;
   DATA[1706,35] := 249.984;
   DATA[1706,36] := 1.681991;
   DATA[1706,37] := 188.8458;
   DATA[1706,38] := 0.000128152;
   DATA[1706,39] := 1.0;
   DATA[1707,1] := 815.3975;
   DATA[1707,2] := 1.0;
   DATA[1707,3] := 1.0;
   DATA[1707,4] := 262.625;
   DATA[1707,5] := 8.46533;
   DATA[1707,6] := 319.6616;
   DATA[1707,8] := 1.0;
   DATA[1707,9] := 1.0;
   DATA[1707,10] := 1.0;
   DATA[1707,11] := 19.79;
   DATA[1707,12] := 2.209653;
   DATA[1707,13] := 851.4243;
   DATA[1707,14] := 1.0;
   DATA[1707,15] := 2.0;
   DATA[1707,16] := 1.0;
   DATA[1707,17] := 1.0;
   DATA[1707,18] := 1.0;
   DATA[1707,19] := 2.0;
   DATA[1707,20] := 148.808;
   DATA[1707,21] := 154.1912;
   DATA[1707,22] := 1.710826;
   DATA[1707,23] := 805.332;
   DATA[1707,24] := 2.0;
   DATA[1707,25] := 2.0;
   DATA[1707,26] := 7.876058;
   DATA[1707,27] := 143.0915;
   DATA[1707,28] := 262.657;
   DATA[1707,29] := 12.11228;
   DATA[1707,30] := 1.723661;
   DATA[1707,31] := 1.276803;
   DATA[1707,32] := 0.7353967;
   DATA[1707,33] := 0.3084905;
   DATA[1707,34] := 2.0;
   DATA[1707,35] := 250.0;
   DATA[1707,36] := 1.681991;
   DATA[1707,37] := 188.8458;
   DATA[1707,38] := 0.000128152;
   DATA[1707,39] := 1.0;
   DATA[1708,1] := 815.3975;
   DATA[1708,2] := 1.0;
   DATA[1708,3] := 1.0;
   DATA[1708,4] := 262.625;
   DATA[1708,5] := 8.46533;
   DATA[1708,6] := 319.6616;
   DATA[1708,8] := 1.0;
   DATA[1708,9] := 1.0;
   DATA[1708,10] := 1.0;
   DATA[1708,11] := 19.79;
   DATA[1708,12] := 2.209653;
   DATA[1708,13] := 850.8235;
   DATA[1708,14] := 1.0;
   DATA[1708,15] := 2.0;
   DATA[1708,16] := 1.0;
   DATA[1708,17] := 1.0;
   DATA[1708,18] := 1.0;
   DATA[1708,19] := 2.0;
   DATA[1708,20] := 148.808;
   DATA[1708,21] := 154.3963;
   DATA[1708,22] := 1.710826;
   DATA[1708,23] := 805.4858;
   DATA[1708,24] := 2.0;
   DATA[1708,25] := 2.0;
   DATA[1708,26] := 7.876058;
   DATA[1708,27] := 143.0915;
   DATA[1708,28] := 262.657;
   DATA[1708,29] := 12.11228;
   DATA[1708,30] := 1.723661;
   DATA[1708,31] := 1.289484;
   DATA[1708,32] := 0.7353967;
   DATA[1708,33] := 0.3084905;
   DATA[1708,34] := 2.0;
   DATA[1708,35] := 250.032;
   DATA[1708,36] := 1.681991;
   DATA[1708,37] := 188.8458;
   DATA[1708,38] := 0.000128152;
   DATA[1708,39] := 1.0;
   DATA[1709,1] := 814.9658;
   DATA[1709,2] := 1.0;
   DATA[1709,3] := 1.0;
   DATA[1709,4] := 262.625;
   DATA[1709,5] := 8.46533;
   DATA[1709,6] := 319.6616;
   DATA[1709,8] := 1.0;
   DATA[1709,9] := 1.0;
   DATA[1709,10] := 1.0;
   DATA[1709,11] := 19.79;
   DATA[1709,12] := 2.209525;
   DATA[1709,13] := 850.6633;
   DATA[1709,14] := 1.0;
   DATA[1709,15] := 2.0;
   DATA[1709,16] := 1.0;
   DATA[1709,17] := 1.0;
   DATA[1709,18] := 1.0;
   DATA[1709,19] := 2.0;
   DATA[1709,20] := 148.808;
   DATA[1709,21] := 154.3963;
   DATA[1709,22] := 1.711979;
   DATA[1709,23] := 805.332;
   DATA[1709,24] := 2.0;
   DATA[1709,25] := 2.0;
   DATA[1709,26] := 7.876058;
   DATA[1709,27] := 143.0915;
   DATA[1709,28] := 262.657;
   DATA[1709,29] := 12.11228;
   DATA[1709,30] := 1.723661;
   DATA[1709,31] := 1.298578;
   DATA[1709,32] := 0.7353967;
   DATA[1709,33] := 0.3084905;
   DATA[1709,34] := 2.0;
   DATA[1709,35] := 250.032;
   DATA[1709,36] := 1.681991;
   DATA[1709,37] := 188.8458;
   DATA[1709,38] := 0.000128152;
   DATA[1709,39] := 1.0;
   DATA[1710,1] := 815.3583;
   DATA[1710,2] := 1.0;
   DATA[1710,3] := 1.0;
   DATA[1710,4] := 262.625;
   DATA[1710,5] := 8.46533;
   DATA[1710,6] := 319.6616;
   DATA[1710,8] := 1.0;
   DATA[1710,9] := 1.0;
   DATA[1710,10] := 1.0;
   DATA[1710,11] := 19.79;
   DATA[1710,12] := 2.209269;
   DATA[1710,13] := 850.0225;
   DATA[1710,14] := 1.0;
   DATA[1710,15] := 2.0;
   DATA[1710,16] := 1.0;
   DATA[1710,17] := 1.0;
   DATA[1710,18] := 1.0;
   DATA[1710,19] := 2.0;
   DATA[1710,20] := 148.808;
   DATA[1710,21] := 154.3963;
   DATA[1710,22] := 1.712748;
   DATA[1710,23] := 805.5627;
   DATA[1710,24] := 2.0;
   DATA[1710,25] := 2.0;
   DATA[1710,26] := 7.876058;
   DATA[1710,27] := 143.0915;
   DATA[1710,28] := 262.657;
   DATA[1710,29] := 12.11228;
   DATA[1710,30] := 1.723661;
   DATA[1710,31] := 1.292558;
   DATA[1710,32] := 0.7353967;
   DATA[1710,33] := 0.3084905;
   DATA[1710,34] := 2.0;
   DATA[1710,35] := 250.032;
   DATA[1710,36] := 1.681991;
   DATA[1710,37] := 188.8458;
   DATA[1710,38] := 0.000128152;
   DATA[1710,39] := 1.0;
   DATA[1711,1] := 815.0835;
   DATA[1711,2] := 1.0;
   DATA[1711,3] := 1.0;
   DATA[1711,4] := 262.625;
   DATA[1711,5] := 8.46533;
   DATA[1711,6] := 319.6616;
   DATA[1711,8] := 1.0;
   DATA[1711,9] := 1.0;
   DATA[1711,10] := 1.0;
   DATA[1711,11] := 19.79;
   DATA[1711,12] := 2.209269;
   DATA[1711,13] := 849.7421;
   DATA[1711,14] := 1.0;
   DATA[1711,15] := 2.0;
   DATA[1711,16] := 1.0;
   DATA[1711,17] := 1.0;
   DATA[1711,18] := 1.0;
   DATA[1711,19] := 2.0;
   DATA[1711,20] := 148.808;
   DATA[1711,21] := 154.3963;
   DATA[1711,22] := 1.712748;
   DATA[1711,23] := 805.6011;
   DATA[1711,24] := 2.0;
   DATA[1711,25] := 2.0;
   DATA[1711,26] := 7.876058;
   DATA[1711,27] := 143.0915;
   DATA[1711,28] := 262.657;
   DATA[1711,29] := 12.11228;
   DATA[1711,30] := 1.723661;
   DATA[1711,31] := 1.283464;
   DATA[1711,32] := 0.7378293;
   DATA[1711,33] := 0.3084905;
   DATA[1711,34] := 2.0;
   DATA[1711,35] := 249.9039;
   DATA[1711,36] := 1.601897;
   DATA[1711,37] := 188.8458;
   DATA[1711,38] := 0.000128152;
   DATA[1711,39] := 1.0;
   DATA[1712,1] := 814.9658;
   DATA[1712,2] := 1.0;
   DATA[1712,3] := 1.0;
   DATA[1712,4] := 262.625;
   DATA[1712,5] := 8.46533;
   DATA[1712,6] := 319.6616;
   DATA[1712,8] := 1.0;
   DATA[1712,9] := 1.0;
   DATA[1712,10] := 1.0;
   DATA[1712,11] := 19.73558;
   DATA[1712,12] := 2.208116;
   DATA[1712,13] := 848.7007;
   DATA[1712,14] := 1.0;
   DATA[1712,15] := 2.0;
   DATA[1712,16] := 1.0;
   DATA[1712,17] := 1.0;
   DATA[1712,18] := 1.0;
   DATA[1712,19] := 2.0;
   DATA[1712,20] := 148.808;
   DATA[1712,21] := 154.3963;
   DATA[1712,22] := 1.712748;
   DATA[1712,23] := 805.9088;
   DATA[1712,24] := 2.0;
   DATA[1712,25] := 2.0;
   DATA[1712,26] := 7.876058;
   DATA[1712,27] := 143.0915;
   DATA[1712,28] := 262.657;
   DATA[1712,29] := 12.11228;
   DATA[1712,30] := 1.723661;
   DATA[1712,31] := 1.27232;
   DATA[1712,32] := 0.7378293;
   DATA[1712,33] := 0.3084905;
   DATA[1712,34] := 2.0;
   DATA[1712,35] := 249.7437;
   DATA[1712,36] := 1.601897;
   DATA[1712,37] := 188.6055;
   DATA[1712,38] := 0.000128152;
   DATA[1712,39] := 1.0;
   DATA[1713,1] := 815.3975;
   DATA[1713,2] := 1.0;
   DATA[1713,3] := 1.0;
   DATA[1713,4] := 262.625;
   DATA[1713,5] := 8.46533;
   DATA[1713,6] := 319.6616;
   DATA[1713,8] := 1.0;
   DATA[1713,9] := 1.0;
   DATA[1713,10] := 1.0;
   DATA[1713,11] := 19.72277;
   DATA[1713,12] := 2.208116;
   DATA[1713,13] := 848.6205;
   DATA[1713,14] := 1.0;
   DATA[1713,15] := 2.0;
   DATA[1713,16] := 1.0;
   DATA[1713,17] := 1.0;
   DATA[1713,18] := 1.0;
   DATA[1713,19] := 2.0;
   DATA[1713,20] := 148.808;
   DATA[1713,21] := 154.3963;
   DATA[1713,22] := 1.712748;
   DATA[1713,23] := 806.0626;
   DATA[1713,24] := 2.0;
   DATA[1713,25] := 2.0;
   DATA[1713,26] := 7.876058;
   DATA[1713,27] := 143.0915;
   DATA[1713,28] := 262.657;
   DATA[1713,29] := 12.11228;
   DATA[1713,30] := 1.723661;
   DATA[1713,31] := 1.276419;
   DATA[1713,32] := 0.7378293;
   DATA[1713,33] := 0.3084905;
   DATA[1713,34] := 2.0;
   DATA[1713,35] := 249.7437;
   DATA[1713,36] := 1.601897;
   DATA[1713,37] := 188.6055;
   DATA[1713,38] := 0.000128152;
   DATA[1713,39] := 1.0;
   DATA[1714,1] := 815.5153;
   DATA[1714,2] := 1.0;
   DATA[1714,3] := 1.0;
   DATA[1714,4] := 262.625;
   DATA[1714,5] := 8.46533;
   DATA[1714,6] := 319.6616;
   DATA[1714,8] := 1.0;
   DATA[1714,9] := 1.0;
   DATA[1714,10] := 1.0;
   DATA[1714,11] := 19.72277;
   DATA[1714,12] := 2.208116;
   DATA[1714,13] := 848.0598;
   DATA[1714,14] := 1.0;
   DATA[1714,15] := 2.0;
   DATA[1714,16] := 1.0;
   DATA[1714,17] := 1.0;
   DATA[1714,18] := 1.0;
   DATA[1714,19] := 2.0;
   DATA[1714,20] := 148.808;
   DATA[1714,21] := 154.3963;
   DATA[1714,22] := 1.712748;
   DATA[1714,23] := 806.1779;
   DATA[1714,24] := 2.0;
   DATA[1714,25] := 2.0;
   DATA[1714,26] := 7.876058;
   DATA[1714,27] := 143.0915;
   DATA[1714,28] := 262.657;
   DATA[1714,29] := 12.11228;
   DATA[1714,30] := 1.723661;
   DATA[1714,31] := 1.276547;
   DATA[1714,32] := 0.7378293;
   DATA[1714,33] := 0.3084905;
   DATA[1714,34] := 2.0;
   DATA[1714,35] := 249.7437;
   DATA[1714,36] := 1.601897;
   DATA[1714,37] := 188.6055;
   DATA[1714,38] := 0.000128152;
   DATA[1714,39] := 1.0;
   DATA[1715,1] := 815.3583;
   DATA[1715,2] := 1.0;
   DATA[1715,3] := 1.0;
   DATA[1715,4] := 262.625;
   DATA[1715,5] := 8.46533;
   DATA[1715,6] := 319.6616;
   DATA[1715,8] := 1.0;
   DATA[1715,9] := 1.0;
   DATA[1715,10] := 1.0;
   DATA[1715,11] := 19.77079;
   DATA[1715,12] := 2.208884;
   DATA[1715,13] := 847.4189;
   DATA[1715,14] := 1.0;
   DATA[1715,15] := 2.0;
   DATA[1715,16] := 1.0;
   DATA[1715,17] := 1.0;
   DATA[1715,18] := 1.0;
   DATA[1715,19] := 2.0;
   DATA[1715,20] := 148.808;
   DATA[1715,21] := 154.3963;
   DATA[1715,22] := 1.712748;
   DATA[1715,23] := 805.9088;
   DATA[1715,24] := 2.0;
   DATA[1715,25] := 2.0;
   DATA[1715,26] := 7.876058;
   DATA[1715,27] := 143.0915;
   DATA[1715,28] := 262.657;
   DATA[1715,29] := 12.11228;
   DATA[1715,30] := 1.721866;
   DATA[1715,31] := 1.262969;
   DATA[1715,32] := 0.7378293;
   DATA[1715,33] := 0.3084905;
   DATA[1715,34] := 2.0;
   DATA[1715,35] := 249.7437;
   DATA[1715,36] := 1.601897;
   DATA[1715,37] := 188.6055;
   DATA[1715,38] := 0.000128152;
   DATA[1715,39] := 1.0;
   DATA[1716,1] := 815.3583;
   DATA[1716,2] := 1.0;
   DATA[1716,3] := 1.0;
   DATA[1716,4] := 262.625;
   DATA[1716,5] := 8.46533;
   DATA[1716,6] := 319.6616;
   DATA[1716,8] := 1.0;
   DATA[1716,9] := 1.0;
   DATA[1716,10] := 1.0;
   DATA[1716,11] := 19.79;
   DATA[1716,12] := 2.209525;
   DATA[1716,13] := 847.0985;
   DATA[1716,14] := 1.0;
   DATA[1716,15] := 2.0;
   DATA[1716,16] := 1.0;
   DATA[1716,17] := 1.0;
   DATA[1716,18] := 1.0;
   DATA[1716,19] := 2.0;
   DATA[1716,20] := 148.808;
   DATA[1716,21] := 154.2938;
   DATA[1716,22] := 1.712748;
   DATA[1716,23] := 806.1779;
   DATA[1716,24] := 2.0;
   DATA[1716,25] := 2.0;
   DATA[1716,26] := 7.876058;
   DATA[1716,27] := 143.0915;
   DATA[1716,28] := 262.657;
   DATA[1716,29] := 12.11228;
   DATA[1716,30] := 1.721738;
   DATA[1716,31] := 1.254259;
   DATA[1716,32] := 0.7378293;
   DATA[1716,33] := 0.3080421;
   DATA[1716,34] := 2.0;
   DATA[1716,35] := 249.7437;
   DATA[1716,36] := 1.601897;
   DATA[1716,37] := 188.6055;
   DATA[1716,38] := 0.000128152;
   DATA[1716,39] := 1.0;
   DATA[1717,1] := 815.319;
   DATA[1717,2] := 1.0;
   DATA[1717,3] := 1.0;
   DATA[1717,4] := 262.625;
   DATA[1717,5] := 8.46533;
   DATA[1717,6] := 319.6616;
   DATA[1717,8] := 1.0;
   DATA[1717,9] := 1.0;
   DATA[1717,10] := 1.0;
   DATA[1717,11] := 19.79;
   DATA[1717,12] := 2.211447;
   DATA[1717,13] := 846.6179;
   DATA[1717,14] := 1.0;
   DATA[1717,15] := 2.0;
   DATA[1717,16] := 1.0;
   DATA[1717,17] := 1.0;
   DATA[1717,18] := 1.0;
   DATA[1717,19] := 2.0;
   DATA[1717,20] := 148.808;
   DATA[1717,21] := 154.2938;
   DATA[1717,22] := 1.71262;
   DATA[1717,23] := 806.1779;
   DATA[1717,24] := 2.0;
   DATA[1717,25] := 2.0;
   DATA[1717,26] := 7.876058;
   DATA[1717,27] := 143.0915;
   DATA[1717,28] := 262.657;
   DATA[1717,29] := 12.11228;
   DATA[1717,30] := 1.721738;
   DATA[1717,31] := 1.257846;
   DATA[1717,32] := 0.7378293;
   DATA[1717,33] := 0.3080421;
   DATA[1717,34] := 2.0;
   DATA[1717,35] := 249.8238;
   DATA[1717,36] := 1.617916;
   DATA[1717,37] := 188.7176;
   DATA[1717,38] := 0.000128152;
   DATA[1717,39] := 1.0;
   DATA[1718,1] := 815.2013;
   DATA[1718,2] := 1.0;
   DATA[1718,3] := 1.0;
   DATA[1718,4] := 262.625;
   DATA[1718,5] := 8.46533;
   DATA[1718,6] := 319.6616;
   DATA[1718,8] := 1.0;
   DATA[1718,9] := 1.0;
   DATA[1718,10] := 1.0;
   DATA[1718,11] := 19.79;
   DATA[1718,12] := 2.211959;
   DATA[1718,13] := 846.6579;
   DATA[1718,14] := 1.0;
   DATA[1718,15] := 2.0;
   DATA[1718,16] := 1.0;
   DATA[1718,17] := 1.0;
   DATA[1718,18] := 1.0;
   DATA[1718,19] := 2.0;
   DATA[1718,20] := 148.808;
   DATA[1718,21] := 154.2938;
   DATA[1718,22] := 1.711338;
   DATA[1718,23] := 806.3702;
   DATA[1718,24] := 2.0;
   DATA[1718,25] := 2.0;
   DATA[1718,26] := 7.876058;
   DATA[1718,27] := 143.0915;
   DATA[1718,28] := 262.657;
   DATA[1718,29] := 12.11228;
   DATA[1718,30] := 1.722763;
   DATA[1718,31] := 1.271679;
   DATA[1718,32] := 0.7357808;
   DATA[1718,33] := 0.3080421;
   DATA[1718,34] := 2.0;
   DATA[1718,35] := 249.8238;
   DATA[1718,36] := 1.617916;
   DATA[1718,37] := 188.7176;
   DATA[1718,38] := 0.000128152;
   DATA[1718,39] := 1.0;
   DATA[1719,1] := 815.162;
   DATA[1719,2] := 1.0;
   DATA[1719,3] := 1.0;
   DATA[1719,4] := 262.625;
   DATA[1719,5] := 8.46533;
   DATA[1719,6] := 319.6616;
   DATA[1719,8] := 1.0;
   DATA[1719,9] := 1.0;
   DATA[1719,10] := 1.0;
   DATA[1719,11] := 19.81881;
   DATA[1719,12] := 2.211959;
   DATA[1719,13] := 846.2974;
   DATA[1719,14] := 1.0;
   DATA[1719,15] := 2.0;
   DATA[1719,16] := 1.0;
   DATA[1719,17] := 1.0;
   DATA[1719,18] := 1.0;
   DATA[1719,19] := 2.0;
   DATA[1719,20] := 148.808;
   DATA[1719,21] := 154.2938;
   DATA[1719,22] := 1.711338;
   DATA[1719,23] := 806.6393;
   DATA[1719,24] := 2.0;
   DATA[1719,25] := 2.0;
   DATA[1719,26] := 7.876058;
   DATA[1719,27] := 143.0915;
   DATA[1719,28] := 262.5288;
   DATA[1719,29] := 12.11228;
   DATA[1719,30] := 1.722892;
   DATA[1719,31] := 1.289612;
   DATA[1719,32] := 0.7352687;
   DATA[1719,33] := 0.3086186;
   DATA[1719,34] := 2.0;
   DATA[1719,35] := 249.8558;
   DATA[1719,36] := 1.617916;
   DATA[1719,37] := 188.7176;
   DATA[1719,38] := 0.000128152;
   DATA[1719,39] := 1.0;
   DATA[1720,1] := 815.319;
   DATA[1720,2] := 1.0;
   DATA[1720,3] := 1.0;
   DATA[1720,4] := 262.625;
   DATA[1720,5] := 8.46533;
   DATA[1720,6] := 319.6616;
   DATA[1720,8] := 1.0;
   DATA[1720,9] := 1.0;
   DATA[1720,10] := 1.0;
   DATA[1720,11] := 19.81881;
   DATA[1720,12] := 2.211959;
   DATA[1720,13] := 846.0171;
   DATA[1720,14] := 1.0;
   DATA[1720,15] := 2.0;
   DATA[1720,16] := 1.0;
   DATA[1720,17] := 1.0;
   DATA[1720,18] := 1.0;
   DATA[1720,19] := 2.0;
   DATA[1720,20] := 148.808;
   DATA[1720,21] := 154.2938;
   DATA[1720,22] := 1.711338;
   DATA[1720,23] := 806.3317;
   DATA[1720,24] := 2.0;
   DATA[1720,25] := 2.0;
   DATA[1720,26] := 7.876058;
   DATA[1720,27] := 143.0915;
   DATA[1720,28] := 262.5288;
   DATA[1720,29] := 12.11228;
   DATA[1720,30] := 1.722892;
   DATA[1720,31] := 1.301524;
   DATA[1720,32] := 0.7352687;
   DATA[1720,33] := 0.3086186;
   DATA[1720,34] := 2.0;
   DATA[1720,35] := 249.9199;
   DATA[1720,36] := 1.617916;
   DATA[1720,37] := 188.7176;
   DATA[1720,38] := 0.000128152;
   DATA[1720,39] := 1.0;
   DATA[1721,1] := 815.162;
   DATA[1721,2] := 1.0;
   DATA[1721,3] := 1.0;
   DATA[1721,4] := 262.625;
   DATA[1721,5] := 8.46533;
   DATA[1721,6] := 319.6616;
   DATA[1721,8] := 1.0;
   DATA[1721,9] := 1.0;
   DATA[1721,10] := 1.0;
   DATA[1721,11] := 19.81881;
   DATA[1721,12] := 2.211959;
   DATA[1721,13] := 845.216;
   DATA[1721,14] := 1.0;
   DATA[1721,15] := 2.0;
   DATA[1721,16] := 1.0;
   DATA[1721,17] := 1.0;
   DATA[1721,18] := 1.0;
   DATA[1721,19] := 2.0;
   DATA[1721,20] := 148.808;
   DATA[1721,21] := 154.2938;
   DATA[1721,22] := 1.711338;
   DATA[1721,23] := 807.0239;
   DATA[1721,24] := 2.0;
   DATA[1721,25] := 2.0;
   DATA[1721,26] := 7.876058;
   DATA[1721,27] := 143.0915;
   DATA[1721,28] := 262.5288;
   DATA[1721,29] := 12.11228;
   DATA[1721,30] := 1.722892;
   DATA[1721,31] := 1.29576;
   DATA[1721,32] := 0.7352687;
   DATA[1721,33] := 0.3086186;
   DATA[1721,34] := 2.0;
   DATA[1721,35] := 249.9199;
   DATA[1721,36] := 1.617916;
   DATA[1721,37] := 188.7176;
   DATA[1721,38] := 0.000128152;
   DATA[1721,39] := 1.0;
   DATA[1722,1] := 815.2013;
   DATA[1722,2] := 1.0;
   DATA[1722,3] := 1.0;
   DATA[1722,4] := 262.625;
   DATA[1722,5] := 8.46533;
   DATA[1722,6] := 319.6616;
   DATA[1722,8] := 1.0;
   DATA[1722,9] := 1.0;
   DATA[1722,10] := 1.0;
   DATA[1722,11] := 19.76759;
   DATA[1722,12] := 2.211959;
   DATA[1722,13] := 845.0958;
   DATA[1722,14] := 1.0;
   DATA[1722,15] := 2.0;
   DATA[1722,16] := 1.0;
   DATA[1722,17] := 1.0;
   DATA[1722,18] := 1.0;
   DATA[1722,19] := 2.0;
   DATA[1722,20] := 148.808;
   DATA[1722,21] := 154.2938;
   DATA[1722,22] := 1.711338;
   DATA[1722,23] := 806.7547;
   DATA[1722,24] := 2.0;
   DATA[1722,25] := 2.0;
   DATA[1722,26] := 7.876058;
   DATA[1722,27] := 143.2453;
   DATA[1722,28] := 262.5288;
   DATA[1722,29] := 12.11228;
   DATA[1722,30] := 1.722892;
   DATA[1722,31] := 1.298194;
   DATA[1722,32] := 0.7352687;
   DATA[1722,33] := 0.3086186;
   DATA[1722,34] := 2.0;
   DATA[1722,35] := 249.9199;
   DATA[1722,36] := 1.617916;
   DATA[1722,37] := 188.7176;
   DATA[1722,38] := 0.000128152;
   DATA[1722,39] := 1.0;
   DATA[1723,1] := 815.2013;
   DATA[1723,2] := 1.0;
   DATA[1723,3] := 1.0;
   DATA[1723,4] := 262.625;
   DATA[1723,5] := 8.46533;
   DATA[1723,6] := 319.6616;
   DATA[1723,8] := 1.0;
   DATA[1723,9] := 1.0;
   DATA[1723,10] := 1.0;
   DATA[1723,11] := 19.70357;
   DATA[1723,12] := 2.210037;
   DATA[1723,13] := 844.455;
   DATA[1723,14] := 1.0;
   DATA[1723,15] := 2.0;
   DATA[1723,16] := 1.0;
   DATA[1723,17] := 1.0;
   DATA[1723,18] := 1.0;
   DATA[1723,19] := 2.0;
   DATA[1723,20] := 148.808;
   DATA[1723,21] := 154.2938;
   DATA[1723,22] := 1.710441;
   DATA[1723,23] := 806.8701;
   DATA[1723,24] := 2.0;
   DATA[1723,25] := 2.0;
   DATA[1723,26] := 7.876058;
   DATA[1723,27] := 143.2453;
   DATA[1723,28] := 262.5288;
   DATA[1723,29] := 12.11228;
   DATA[1723,30] := 1.722892;
   DATA[1723,31] := 1.292686;
   DATA[1723,32] := 0.7352687;
   DATA[1723,33] := 0.3086186;
   DATA[1723,34] := 2.0;
   DATA[1723,35] := 249.9199;
   DATA[1723,36] := 1.617916;
   DATA[1723,37] := 188.7176;
   DATA[1723,38] := 0.000128152;
   DATA[1723,39] := 1.0;
   DATA[1724,1] := 815.005;
   DATA[1724,2] := 1.0;
   DATA[1724,3] := 1.0;
   DATA[1724,4] := 262.625;
   DATA[1724,5] := 8.46533;
   DATA[1724,6] := 319.6616;
   DATA[1724,8] := 1.0;
   DATA[1724,9] := 1.0;
   DATA[1724,10] := 1.0;
   DATA[1724,11] := 19.69076;
   DATA[1724,12] := 2.209525;
   DATA[1724,13] := 844.0945;
   DATA[1724,14] := 1.0;
   DATA[1724,15] := 2.0;
   DATA[1724,16] := 1.0;
   DATA[1724,17] := 1.0;
   DATA[1724,18] := 1.0;
   DATA[1724,19] := 2.0;
   DATA[1724,20] := 148.808;
   DATA[1724,21] := 154.2938;
   DATA[1724,22] := 1.710441;
   DATA[1724,23] := 806.7547;
   DATA[1724,24] := 2.0;
   DATA[1724,25] := 2.0;
   DATA[1724,26] := 7.876058;
   DATA[1724,27] := 143.2453;
   DATA[1724,28] := 262.5288;
   DATA[1724,29] := 12.11228;
   DATA[1724,30] := 1.721482;
   DATA[1724,31] := 1.290893;
   DATA[1724,32] := 0.7352687;
   DATA[1724,33] := 0.3086186;
   DATA[1724,34] := 2.0;
   DATA[1724,35] := 249.7116;
   DATA[1724,36] := 1.617916;
   DATA[1724,37] := 188.7176;
   DATA[1724,38] := 0.000128152;
   DATA[1724,39] := 1.0;
   DATA[1725,1] := 814.8873;
   DATA[1725,2] := 1.0;
   DATA[1725,3] := 1.0;
   DATA[1725,4] := 262.625;
   DATA[1725,5] := 8.46533;
   DATA[1725,6] := 319.6616;
   DATA[1725,8] := 1.0;
   DATA[1725,9] := 1.0;
   DATA[1725,10] := 1.0;
   DATA[1725,11] := 19.69076;
   DATA[1725,12] := 2.209397;
   DATA[1725,13] := 843.6539;
   DATA[1725,14] := 1.0;
   DATA[1725,15] := 2.0;
   DATA[1725,16] := 1.0;
   DATA[1725,17] := 1.0;
   DATA[1725,18] := 1.0;
   DATA[1725,19] := 2.0;
   DATA[1725,20] := 148.808;
   DATA[1725,21] := 154.4219;
   DATA[1725,22] := 1.710441;
   DATA[1725,23] := 806.8701;
   DATA[1725,24] := 2.0;
   DATA[1725,25] := 2.0;
   DATA[1725,26] := 7.876058;
   DATA[1725,27] := 143.2453;
   DATA[1725,28] := 262.5288;
   DATA[1725,29] := 12.11228;
   DATA[1725,30] := 1.721482;
   DATA[1725,31] := 1.282183;
   DATA[1725,32] := 0.7352687;
   DATA[1725,33] := 0.3080421;
   DATA[1725,34] := 2.0;
   DATA[1725,35] := 249.6956;
   DATA[1725,36] := 1.617916;
   DATA[1725,37] := 188.5254;
   DATA[1725,38] := 0.000128152;
   DATA[1725,39] := 1.0;
   DATA[1726,1] := 814.9265;
   DATA[1726,2] := 1.0;
   DATA[1726,3] := 1.0;
   DATA[1726,4] := 262.625;
   DATA[1726,5] := 8.46533;
   DATA[1726,6] := 319.6616;
   DATA[1726,8] := 1.0;
   DATA[1726,9] := 1.0;
   DATA[1726,10] := 1.0;
   DATA[1726,11] := 19.74838;
   DATA[1726,12] := 2.208372;
   DATA[1726,13] := 843.013;
   DATA[1726,14] := 1.0;
   DATA[1726,15] := 2.0;
   DATA[1726,16] := 1.0;
   DATA[1726,17] := 1.0;
   DATA[1726,18] := 1.0;
   DATA[1726,19] := 2.0;
   DATA[1726,20] := 148.808;
   DATA[1726,21] := 154.4219;
   DATA[1726,22] := 1.710441;
   DATA[1726,23] := 807.4853;
   DATA[1726,24] := 2.0;
   DATA[1726,25] := 2.0;
   DATA[1726,26] := 7.876058;
   DATA[1726,27] := 143.2453;
   DATA[1726,28] := 262.5288;
   DATA[1726,29] := 12.11228;
   DATA[1726,30] := 1.721482;
   DATA[1726,31] := 1.281286;
   DATA[1726,32] := 0.7352687;
   DATA[1726,33] := 0.3080421;
   DATA[1726,34] := 2.0;
   DATA[1726,35] := 249.6956;
   DATA[1726,36] := 1.617916;
   DATA[1726,37] := 188.5254;
   DATA[1726,38] := 0.000128152;
   DATA[1726,39] := 1.0;
   DATA[1727,1] := 815.319;
   DATA[1727,2] := 1.0;
   DATA[1727,3] := 1.0;
   DATA[1727,4] := 262.625;
   DATA[1727,5] := 8.46533;
   DATA[1727,6] := 319.7385;
   DATA[1727,8] := 1.0;
   DATA[1727,9] := 1.0;
   DATA[1727,10] := 1.0;
   DATA[1727,11] := 19.74838;
   DATA[1727,12] := 2.207603;
   DATA[1727,13] := 842.9329;
   DATA[1727,14] := 1.0;
   DATA[1727,15] := 2.0;
   DATA[1727,16] := 1.0;
   DATA[1727,17] := 1.0;
   DATA[1727,18] := 1.0;
   DATA[1727,19] := 2.0;
   DATA[1727,20] := 148.808;
   DATA[1727,21] := 154.4219;
   DATA[1727,22] := 1.710441;
   DATA[1727,23] := 807.6775;
   DATA[1727,24] := 2.0;
   DATA[1727,25] := 2.0;
   DATA[1727,26] := 7.876058;
   DATA[1727,27] := 143.2453;
   DATA[1727,28] := 262.5288;
   DATA[1727,29] := 12.11228;
   DATA[1727,30] := 1.721482;
   DATA[1727,31] := 1.291149;
   DATA[1727,32] := 0.7352687;
   DATA[1727,33] := 0.3080421;
   DATA[1727,34] := 2.0;
   DATA[1727,35] := 249.6956;
   DATA[1727,36] := 1.617916;
   DATA[1727,37] := 188.5254;
   DATA[1727,38] := 0.000128152;
   DATA[1727,39] := 1.0;
   DATA[1728,1] := 815.5546;
   DATA[1728,2] := 1.0;
   DATA[1728,3] := 1.0;
   DATA[1728,4] := 262.625;
   DATA[1728,5] := 8.463408;
   DATA[1728,6] := 319.7385;
   DATA[1728,8] := 1.0;
   DATA[1728,9] := 1.0;
   DATA[1728,10] := 1.0;
   DATA[1728,11] := 19.74838;
   DATA[1728,12] := 2.207603;
   DATA[1728,13] := 842.212;
   DATA[1728,14] := 1.0;
   DATA[1728,15] := 2.0;
   DATA[1728,16] := 1.0;
   DATA[1728,17] := 1.0;
   DATA[1728,18] := 1.0;
   DATA[1728,19] := 2.0;
   DATA[1728,20] := 148.808;
   DATA[1728,21] := 154.4219;
   DATA[1728,22] := 1.710441;
   DATA[1728,23] := 807.639;
   DATA[1728,24] := 2.0;
   DATA[1728,25] := 2.0;
   DATA[1728,26] := 7.876058;
   DATA[1728,27] := 143.1172;
   DATA[1728,28] := 262.5288;
   DATA[1728,29] := 12.11228;
   DATA[1728,30] := 1.721482;
   DATA[1728,31] := 1.286025;
   DATA[1728,32] := 0.7352687;
   DATA[1728,33] := 0.3080421;
   DATA[1728,34] := 2.0;
   DATA[1728,35] := 249.6956;
   DATA[1728,36] := 1.617916;
   DATA[1728,37] := 188.5254;
   DATA[1728,38] := 0.000128152;
   DATA[1728,39] := 1.0;
   DATA[1729,1] := 815.5938;
   DATA[1729,2] := 1.0;
   DATA[1729,3] := 1.0;
   DATA[1729,4] := 262.625;
   DATA[1729,5] := 8.463408;
   DATA[1729,6] := 319.7385;
   DATA[1729,8] := 1.0;
   DATA[1729,9] := 1.0;
   DATA[1729,10] := 1.0;
   DATA[1729,11] := 19.74838;
   DATA[1729,12] := 2.207603;
   DATA[1729,13] := 842.252;
   DATA[1729,14] := 1.0;
   DATA[1729,15] := 2.0;
   DATA[1729,16] := 1.0;
   DATA[1729,17] := 1.0;
   DATA[1729,18] := 1.0;
   DATA[1729,19] := 2.0;
   DATA[1729,20] := 148.808;
   DATA[1729,21] := 154.4219;
   DATA[1729,22] := 1.710954;
   DATA[1729,23] := 808.062;
   DATA[1729,24] := 2.0;
   DATA[1729,25] := 2.0;
   DATA[1729,26] := 7.876058;
   DATA[1729,27] := 143.1172;
   DATA[1729,28] := 262.5288;
   DATA[1729,29] := 12.11228;
   DATA[1729,30] := 1.721482;
   DATA[1729,31] := 1.281927;
   DATA[1729,32] := 0.7352687;
   DATA[1729,33] := 0.3083624;
   DATA[1729,34] := 2.0;
   DATA[1729,35] := 249.6956;
   DATA[1729,36] := 1.617916;
   DATA[1729,37] := 188.7016;
   DATA[1729,38] := 0.000128152;
   DATA[1729,39] := 1.0;
   DATA[1730,1] := 815.162;
   DATA[1730,3] := 1.0;
   DATA[1730,4] := 262.625;
   DATA[1730,5] := 8.463408;
   DATA[1730,6] := 319.7385;
   DATA[1730,8] := 1.0;
   DATA[1730,9] := 1.0;
   DATA[1730,10] := 1.0;
   DATA[1730,11] := 19.73558;
   DATA[1730,12] := 2.208628;
   DATA[1730,13] := 841.2907;
   DATA[1730,14] := 1.0;
   DATA[1730,15] := 2.0;
   DATA[1730,16] := 1.0;
   DATA[1730,17] := 1.0;
   DATA[1730,18] := 1.0;
   DATA[1730,19] := 2.0;
   DATA[1730,20] := 148.808;
   DATA[1730,21] := 154.4219;
   DATA[1730,22] := 1.710954;
   DATA[1730,23] := 807.4853;
   DATA[1730,24] := 2.0;
   DATA[1730,25] := 2.0;
   DATA[1730,26] := 7.876058;
   DATA[1730,27] := 143.1172;
   DATA[1730,28] := 262.5288;
   DATA[1730,29] := 12.11228;
   DATA[1730,30] := 1.721866;
   DATA[1730,31] := 1.281927;
   DATA[1730,32] := 0.7352687;
   DATA[1730,33] := 0.3083624;
   DATA[1730,34] := 2.0;
   DATA[1730,35] := 249.6956;
   DATA[1730,36] := 1.617916;
   DATA[1730,37] := 188.7016;
   DATA[1730,38] := 0.000128152;
   DATA[1730,39] := 1.0;
   DATA[1731,1] := 815.2013;
   DATA[1731,3] := 1.0;
   DATA[1731,4] := 262.625;
   DATA[1731,5] := 8.463408;
   DATA[1731,6] := 319.7385;
   DATA[1731,8] := 1.0;
   DATA[1731,9] := 1.0;
   DATA[1731,10] := 1.0;
   DATA[1731,11] := 19.73558;
   DATA[1731,12] := 2.208628;
   DATA[1731,13] := 841.1305;
   DATA[1731,14] := 1.0;
   DATA[1731,15] := 2.0;
   DATA[1731,16] := 1.0;
   DATA[1731,17] := 1.0;
   DATA[1731,18] := 1.0;
   DATA[1731,19] := 2.0;
   DATA[1731,20] := 148.808;
   DATA[1731,21] := 154.4219;
   DATA[1731,22] := 1.710954;
   DATA[1731,23] := 807.5237;
   DATA[1731,24] := 2.0;
   DATA[1731,25] := 2.0;
   DATA[1731,26] := 7.876058;
   DATA[1731,27] := 143.1172;
   DATA[1731,28] := 262.5288;
   DATA[1731,29] := 12.11228;
   DATA[1731,30] := 1.722123;
   DATA[1731,31] := 1.272704;
   DATA[1731,32] := 0.7352687;
   DATA[1731,33] := 0.3083624;
   DATA[1731,34] := 2.0;
   DATA[1731,35] := 249.8718;
   DATA[1731,36] := 1.617916;
   DATA[1731,37] := 188.7016;
   DATA[1731,38] := 0.000128152;
   DATA[1731,39] := 1.0;
   DATA[1732,1] := 815.3975;
   DATA[1732,3] := 1.0;
   DATA[1732,4] := 262.625;
   DATA[1732,5] := 8.466612;
   DATA[1732,6] := 319.7385;
   DATA[1732,8] := 1.0;
   DATA[1732,9] := 1.0;
   DATA[1732,10] := 1.0;
   DATA[1732,11] := 19.77079;
   DATA[1732,12] := 2.209397;
   DATA[1732,13] := 840.4496;
   DATA[1732,14] := 1.0;
   DATA[1732,15] := 2.0;
   DATA[1732,16] := 1.0;
   DATA[1732,17] := 1.0;
   DATA[1732,18] := 1.0;
   DATA[1732,19] := 2.0;
   DATA[1732,20] := 148.808;
   DATA[1732,21] := 154.4219;
   DATA[1732,22] := 1.710954;
   DATA[1732,23] := 807.9082;
   DATA[1732,24] := 2.0;
   DATA[1732,25] := 2.0;
   DATA[1732,26] := 7.876058;
   DATA[1732,27] := 143.1172;
   DATA[1732,28] := 262.5288;
   DATA[1732,29] := 12.11228;
   DATA[1732,30] := 1.722123;
   DATA[1732,31] := 1.281542;
   DATA[1732,32] := 0.7352687;
   DATA[1732,33] := 0.3083624;
   DATA[1732,34] := 2.0;
   DATA[1732,35] := 249.9199;
   DATA[1732,36] := 1.617916;
   DATA[1732,37] := 188.7016;
   DATA[1732,38] := 0.000128152;
   DATA[1732,39] := 1.0;
   DATA[1733,1] := 815.319;
   DATA[1733,3] := 1.0;
   DATA[1733,4] := 262.625;
   DATA[1733,5] := 8.466612;
   DATA[1733,6] := 319.7385;
   DATA[1733,8] := 1.0;
   DATA[1733,9] := 1.0;
   DATA[1733,10] := 1.0;
   DATA[1733,11] := 19.7868;
   DATA[1733,12] := 2.209397;
   DATA[1733,13] := 840.5297;
   DATA[1733,14] := 1.0;
   DATA[1733,15] := 2.0;
   DATA[1733,16] := 1.0;
   DATA[1733,17] := 1.0;
   DATA[1733,18] := 1.0;
   DATA[1733,19] := 2.0;
   DATA[1733,20] := 148.808;
   DATA[1733,21] := 154.4219;
   DATA[1733,22] := 1.710954;
   DATA[1733,23] := 808.2927;
   DATA[1733,24] := 2.0;
   DATA[1733,25] := 2.0;
   DATA[1733,26] := 7.876058;
   DATA[1733,27] := 143.194;
   DATA[1733,28] := 262.5288;
   DATA[1733,29] := 12.11228;
   DATA[1733,30] := 1.722123;
   DATA[1733,31] := 1.299219;
   DATA[1733,32] := 0.7352687;
   DATA[1733,33] := 0.3083624;
   DATA[1733,34] := 2.0;
   DATA[1733,35] := 249.9199;
   DATA[1733,36] := 1.617916;
   DATA[1733,37] := 188.7016;
   DATA[1733,38] := 0.000128152;
   DATA[1733,39] := 1.0;
   DATA[1734,0] := 0.008006917;
   DATA[1734,1] := 814.7695;
   DATA[1734,3] := 1.0;
   DATA[1734,4] := 262.625;
   DATA[1734,5] := 8.466612;
   DATA[1734,6] := 319.7385;
   DATA[1734,8] := 1.0;
   DATA[1734,9] := 1.0;
   DATA[1734,10] := 1.0;
   DATA[1734,11] := 19.7868;
   DATA[1734,12] := 2.209397;
   DATA[1734,13] := 839.4082;
   DATA[1734,14] := 1.0;
   DATA[1734,15] := 2.0;
   DATA[1734,16] := 1.0;
   DATA[1734,17] := 1.0;
   DATA[1734,18] := 1.0;
   DATA[1734,19] := 2.0;
   DATA[1734,20] := 148.808;
   DATA[1734,21] := 154.4219;
   DATA[1734,22] := 1.710954;
   DATA[1734,23] := 808.2158;
   DATA[1734,24] := 2.0;
   DATA[1734,25] := 2.0;
   DATA[1734,26] := 7.876058;
   DATA[1734,27] := 143.3479;
   DATA[1734,28] := 262.5288;
   DATA[1734,29] := 12.11228;
   DATA[1734,30] := 1.722123;
   DATA[1734,31] := 1.305239;
   DATA[1734,32] := 0.7352687;
   DATA[1734,33] := 0.3083624;
   DATA[1734,34] := 2.0;
   DATA[1734,35] := 250.0;
   DATA[1734,36] := 1.665972;
   DATA[1734,37] := 188.7657;
   DATA[1734,38] := 0.000128152;
   DATA[1734,39] := 1.0;
   DATA[1735,0] := 0.08775582;
   DATA[1735,1] := 814.5732;
   DATA[1735,3] := 1.0;
   DATA[1735,4] := 262.625;
   DATA[1735,5] := 8.466612;
   DATA[1735,6] := 319.7385;
   DATA[1735,8] := 1.0;
   DATA[1735,9] := 1.0;
   DATA[1735,10] := 1.0;
   DATA[1735,11] := 19.7868;
   DATA[1735,12] := 2.209397;
   DATA[1735,13] := 839.3281;
   DATA[1735,14] := 1.0;
   DATA[1735,15] := 2.0;
   DATA[1735,16] := 1.0;
   DATA[1735,17] := 1.0;
   DATA[1735,18] := 1.0;
   DATA[1735,19] := 2.0;
   DATA[1735,20] := 148.808;
   DATA[1735,21] := 154.4219;
   DATA[1735,22] := 1.710954;
   DATA[1735,23] := 808.485;
   DATA[1735,24] := 2.0;
   DATA[1735,25] := 2.0;
   DATA[1735,26] := 7.876058;
   DATA[1735,27] := 143.3479;
   DATA[1735,28] := 262.5288;
   DATA[1735,29] := 12.11228;
   DATA[1735,30] := 1.723661;
   DATA[1735,31] := 1.320097;
   DATA[1735,32] := 0.7352687;
   DATA[1735,33] := 0.3083624;
   DATA[1735,34] := 2.0;
   DATA[1735,35] := 250.0;
   DATA[1735,36] := 1.762086;
   DATA[1735,37] := 188.7977;
   DATA[1735,38] := 0.000128152;
   DATA[1735,39] := 1.0;
   DATA[1736,0] := 0.2783205;
   DATA[1736,1] := 814.4948;
   DATA[1736,3] := 1.0;
   DATA[1736,4] := 262.625;
   DATA[1736,5] := 8.46533;
   DATA[1736,6] := 319.7385;
   DATA[1736,8] := 1.0;
   DATA[1736,9] := 1.0;
   DATA[1736,10] := 1.0;
   DATA[1736,11] := 19.76439;
   DATA[1736,12] := 2.209397;
   DATA[1736,13] := 839.1278;
   DATA[1736,14] := 1.0;
   DATA[1736,15] := 2.0;
   DATA[1736,16] := 1.0;
   DATA[1736,17] := 1.0;
   DATA[1736,18] := 1.0;
   DATA[1736,19] := 2.0;
   DATA[1736,20] := 148.808;
   DATA[1736,21] := 154.4219;
   DATA[1736,22] := 1.710826;
   DATA[1736,23] := 808.5619;
   DATA[1736,24] := 2.0;
   DATA[1736,25] := 2.0;
   DATA[1736,26] := 7.876058;
   DATA[1736,27] := 143.3479;
   DATA[1736,28] := 262.5288;
   DATA[1736,29] := 12.11228;
   DATA[1736,30] := 1.724814;
   DATA[1736,31] := 1.306648;
   DATA[1736,32] := 0.7352687;
   DATA[1736,33] := 0.3083624;
   DATA[1736,34] := 2.0;
   DATA[1736,35] := 250.0;
   DATA[1736,36] := 1.762086;
   DATA[1736,37] := 188.7977;
   DATA[1736,38] := 0.000128152;
   DATA[1736,39] := 1.0;
   DATA[1737,0] := 0.554399;
   DATA[1737,1] := 814.4948;
   DATA[1737,3] := 1.0;
   DATA[1737,4] := 262.625;
   DATA[1737,5] := 8.463408;
   DATA[1737,6] := 319.7385;
   DATA[1737,8] := 1.0;
   DATA[1737,9] := 1.0;
   DATA[1737,10] := 1.0;
   DATA[1737,11] := 19.76439;
   DATA[1737,12] := 2.209397;
   DATA[1737,13] := 838.2867;
   DATA[1737,14] := 1.0;
   DATA[1737,15] := 2.0;
   DATA[1737,16] := 1.0;
   DATA[1737,17] := 1.0;
   DATA[1737,18] := 1.0;
   DATA[1737,19] := 2.0;
   DATA[1737,20] := 148.808;
   DATA[1737,21] := 154.4219;
   DATA[1737,22] := 1.709544;
   DATA[1737,23] := 808.3696;
   DATA[1737,24] := 2.0;
   DATA[1737,25] := 2.0;
   DATA[1737,26] := 7.876058;
   DATA[1737,27] := 143.3479;
   DATA[1737,28] := 262.5288;
   DATA[1737,29] := 12.11228;
   DATA[1737,30] := 1.72507;
   DATA[1737,31] := 1.287306;
   DATA[1737,32] := 0.7352687;
   DATA[1737,33] := 0.3083624;
   DATA[1737,34] := 2.0;
   DATA[1737,35] := 250.0;
   DATA[1737,36] := 1.762086;
   DATA[1737,37] := 188.7977;
   DATA[1737,38] := 0.000128152;
   DATA[1737,39] := 1.0;
   DATA[1738,0] := 0.9211158;
   DATA[1738,1] := 814.5732;
   DATA[1738,2] := 2.0;
   DATA[1738,3] := 1.0;
   DATA[1738,4] := 262.625;
   DATA[1738,5] := 8.463408;
   DATA[1738,6] := 319.7385;
   DATA[1738,8] := 1.0;
   DATA[1738,9] := 1.0;
   DATA[1738,10] := 1.0;
   DATA[1738,11] := 19.76439;
   DATA[1738,12] := 2.209397;
   DATA[1738,13] := 837.6859;
   DATA[1738,14] := 1.0;
   DATA[1738,15] := 2.0;
   DATA[1738,16] := 1.0;
   DATA[1738,17] := 1.0;
   DATA[1738,18] := 1.0;
   DATA[1738,19] := 2.0;
   DATA[1738,20] := 148.808;
   DATA[1738,21] := 154.4219;
   DATA[1738,22] := 1.709544;
   DATA[1738,23] := 808.485;
   DATA[1738,24] := 2.0;
   DATA[1738,25] := 2.0;
   DATA[1738,26] := 7.876058;
   DATA[1738,27] := 143.3479;
   DATA[1738,28] := 262.5288;
   DATA[1738,29] := 12.11228;
   DATA[1738,30] := 1.72507;
   DATA[1738,31] := 1.277315;
   DATA[1738,32] := 0.7352687;
   DATA[1738,33] := 0.3083624;
   DATA[1738,34] := 2.0;
   DATA[1738,35] := 250.0;
   DATA[1738,36] := 1.762086;
   DATA[1738,37] := 188.7977;
   DATA[1738,38] := 0.000128152;
   DATA[1738,39] := 1.0;
   DATA[1739,0] := 1.323063;
   DATA[1739,1] := 814.4948;
   DATA[1739,2] := 2.0;
   DATA[1739,3] := 1.0;
   DATA[1739,4] := 262.625;
   DATA[1739,5] := 8.463408;
   DATA[1739,6] := 319.7385;
   DATA[1739,8] := 1.0;
   DATA[1739,9] := 1.0;
   DATA[1739,10] := 1.0;
   DATA[1739,11] := 19.72598;
   DATA[1739,12] := 2.209397;
   DATA[1739,13] := 837.2853;
   DATA[1739,14] := 1.0;
   DATA[1739,15] := 2.0;
   DATA[1739,16] := 1.0;
   DATA[1739,17] := 1.0;
   DATA[1739,18] := 1.0;
   DATA[1739,19] := 2.0;
   DATA[1739,20] := 148.808;
   DATA[1739,21] := 154.3707;
   DATA[1739,22] := 1.710954;
   DATA[1739,23] := 808.4081;
   DATA[1739,24] := 2.0;
   DATA[1739,25] := 2.0;
   DATA[1739,26] := 7.876058;
   DATA[1739,27] := 143.3479;
   DATA[1739,28] := 262.5288;
   DATA[1739,29] := 12.11228;
   DATA[1739,30] := 1.72507;
   DATA[1739,31] := 1.264891;
   DATA[1739,32] := 0.7352687;
   DATA[1739,33] := 0.3083624;
   DATA[1739,34] := 2.0;
   DATA[1739,35] := 250.0;
   DATA[1739,36] := 1.681991;
   DATA[1739,37] := 188.7977;
   DATA[1739,38] := 0.000128152;
   DATA[1739,39] := 1.0;
   DATA[1740,0] := 1.614835;
   DATA[1740,1] := 814.4948;
   DATA[1740,2] := 2.0;
   DATA[1740,3] := 1.0;
   DATA[1740,4] := 262.625;
   DATA[1740,5] := 8.463408;
   DATA[1740,6] := 319.7385;
   DATA[1740,8] := 1.0;
   DATA[1740,9] := 1.0;
   DATA[1740,10] := 1.0;
   DATA[1740,11] := 19.72598;
   DATA[1740,12] := 2.209397;
   DATA[1740,13] := 836.9649;
   DATA[1740,14] := 1.0;
   DATA[1740,15] := 2.0;
   DATA[1740,16] := 1.0;
   DATA[1740,17] := 1.0;
   DATA[1740,18] := 1.0;
   DATA[1740,19] := 2.0;
   DATA[1740,20] := 148.808;
   DATA[1740,21] := 154.3707;
   DATA[1740,22] := 1.711595;
   DATA[1740,23] := 808.2927;
   DATA[1740,24] := 2.0;
   DATA[1740,25] := 2.0;
   DATA[1740,26] := 7.876058;
   DATA[1740,27] := 143.194;
   DATA[1740,28] := 262.5288;
   DATA[1740,29] := 12.11228;
   DATA[1740,30] := 1.724045;
   DATA[1740,31] := 1.272832;
   DATA[1740,32] := 0.7352687;
   DATA[1740,33] := 0.3083624;
   DATA[1740,34] := 2.0;
   DATA[1740,35] := 250.0;
   DATA[1740,36] := 1.681991;
   DATA[1740,37] := 188.7977;
   DATA[1740,38] := 0.000128152;
   DATA[1740,39] := 1.0;
   DATA[1741,0] := 1.958492;
   DATA[1741,1] := 814.377;
   DATA[1741,2] := 2.0;
   DATA[1741,3] := 1.0;
   DATA[1741,4] := 262.625;
   DATA[1741,5] := 8.463408;
   DATA[1741,6] := 319.7385;
   DATA[1741,8] := 1.0;
   DATA[1741,9] := 1.0;
   DATA[1741,10] := 1.0;
   DATA[1741,11] := 19.76439;
   DATA[1741,12] := 2.209397;
   DATA[1741,13] := 836.3641;
   DATA[1741,14] := 1.0;
   DATA[1741,15] := 2.0;
   DATA[1741,16] := 1.0;
   DATA[1741,17] := 1.0;
   DATA[1741,18] := 1.0;
   DATA[1741,19] := 2.0;
   DATA[1741,20] := 148.808;
   DATA[1741,21] := 154.3707;
   DATA[1741,22] := 1.711595;
   DATA[1741,23] := 808.9849;
   DATA[1741,24] := 2.0;
   DATA[1741,25] := 2.0;
   DATA[1741,26] := 7.876058;
   DATA[1741,27] := 143.194;
   DATA[1741,28] := 262.5288;
   DATA[1741,29] := 12.11228;
   DATA[1741,30] := 1.723661;
   DATA[1741,31] := 1.287691;
   DATA[1741,32] := 0.7352687;
   DATA[1741,33] := 0.3083624;
   DATA[1741,34] := 2.0;
   DATA[1741,35] := 250.0;
   DATA[1741,36] := 1.681991;
   DATA[1741,37] := 188.7977;
   DATA[1741,38] := 0.000128152;
   DATA[1741,39] := 1.0;
   DATA[1742,0] := 2.198059;
   DATA[1742,1] := 814.6125;
   DATA[1742,2] := 2.0;
   DATA[1742,3] := 1.0;
   DATA[1742,4] := 262.625;
   DATA[1742,5] := 8.463408;
   DATA[1742,6] := 319.7385;
   DATA[1742,8] := 1.0;
   DATA[1742,9] := 1.0;
   DATA[1742,10] := 1.0;
   DATA[1742,11] := 19.76759;
   DATA[1742,12] := 2.209397;
   DATA[1742,13] := 836.0837;
   DATA[1742,14] := 1.0;
   DATA[1742,15] := 2.0;
   DATA[1742,16] := 1.0;
   DATA[1742,17] := 1.0;
   DATA[1742,18] := 1.0;
   DATA[1742,19] := 2.0;
   DATA[1742,20] := 148.808;
   DATA[1742,21] := 154.3707;
   DATA[1742,22] := 1.711595;
   DATA[1742,23] := 809.4078;
   DATA[1742,24] := 2.0;
   DATA[1742,25] := 2.0;
   DATA[1742,26] := 7.876058;
   DATA[1742,27] := 143.194;
   DATA[1742,28] := 262.5288;
   DATA[1742,29] := 12.11228;
   DATA[1742,30] := 1.723661;
   DATA[1742,31] := 1.280646;
   DATA[1742,32] := 0.7352687;
   DATA[1742,33] := 0.3083624;
   DATA[1742,34] := 2.0;
   DATA[1742,35] := 250.0;
   DATA[1742,36] := 1.681991;
   DATA[1742,37] := 188.7977;
   DATA[1742,38] := 0.000128152;
   DATA[1742,39] := 1.0;
   DATA[1743,0] := 2.335138;
   DATA[1743,1] := 814.534;
   DATA[1743,2] := 2.0;
   DATA[1743,3] := 1.0;
   DATA[1743,4] := 262.625;
   DATA[1743,5] := 8.463408;
   DATA[1743,6] := 319.7385;
   DATA[1743,8] := 1.0;
   DATA[1743,9] := 1.0;
   DATA[1743,10] := 1.0;
   DATA[1743,11] := 19.76759;
   DATA[1743,12] := 2.209397;
   DATA[1743,13] := 835.8033;
   DATA[1743,14] := 1.0;
   DATA[1743,15] := 2.0;
   DATA[1743,16] := 1.0;
   DATA[1743,17] := 1.0;
   DATA[1743,18] := 1.0;
   DATA[1743,19] := 2.0;
   DATA[1743,20] := 148.808;
   DATA[1743,21] := 154.3707;
   DATA[1743,22] := 1.711595;
   DATA[1743,23] := 809.4078;
   DATA[1743,24] := 2.0;
   DATA[1743,25] := 2.0;
   DATA[1743,26] := 7.876058;
   DATA[1743,27] := 143.194;
   DATA[1743,28] := 262.5288;
   DATA[1743,29] := 12.11228;
   DATA[1743,30] := 1.723661;
   DATA[1743,31] := 1.280646;
   DATA[1743,32] := 0.7352687;
   DATA[1743,33] := 0.3083624;
   DATA[1743,34] := 2.0;
   DATA[1743,35] := 250.0;
   DATA[1743,36] := 1.681991;
   DATA[1743,37] := 188.7977;
   DATA[1743,38] := 0.000128152;
   DATA[1743,39] := 1.0;
   DATA[1744,0] := 2.428338;
   DATA[1744,1] := 814.691;
   DATA[1744,2] := 2.0;
   DATA[1744,3] := 1.0;
   DATA[1744,4] := 262.625;
   DATA[1744,5] := 8.463728;
   DATA[1744,6] := 319.7385;
   DATA[1744,8] := 1.0;
   DATA[1744,9] := 1.0;
   DATA[1744,10] := 1.0;
   DATA[1744,11] := 19.76759;
   DATA[1744,12] := 2.209397;
   DATA[1744,13] := 835.8033;
   DATA[1744,14] := 1.0;
   DATA[1744,15] := 2.0;
   DATA[1744,16] := 1.0;
   DATA[1744,17] := 1.0;
   DATA[1744,18] := 1.0;
   DATA[1744,19] := 2.0;
   DATA[1744,20] := 148.808;
   DATA[1744,21] := 154.3707;
   DATA[1744,22] := 1.711595;
   DATA[1744,23] := 809.3309;
   DATA[1744,24] := 2.0;
   DATA[1744,25] := 2.0;
   DATA[1744,26] := 7.876058;
   DATA[1744,27] := 143.194;
   DATA[1744,28] := 262.5288;
   DATA[1744,29] := 12.11228;
   DATA[1744,30] := 1.72302;
   DATA[1744,31] := 1.280646;
   DATA[1744,32] := 0.7352687;
   DATA[1744,33] := 0.3083624;
   DATA[1744,34] := 2.0;
   DATA[1744,35] := 250.0;
   DATA[1744,36] := 1.681991;
   DATA[1744,37] := 188.7977;
   DATA[1744,38] := 0.000128152;
   DATA[1744,39] := 1.0;
   DATA[1745,0] := 2.477981;
   DATA[1745,1] := 814.8088;
   DATA[1745,2] := 2.0;
   DATA[1745,3] := 1.0;
   DATA[1745,4] := 262.625;
   DATA[1745,5] := 8.46501;
   DATA[1745,6] := 319.7385;
   DATA[1745,8] := 1.0;
   DATA[1745,9] := 1.0;
   DATA[1745,10] := 1.0;
   DATA[1745,11] := 19.73878;
   DATA[1745,12] := 2.209397;
   DATA[1745,13] := 835.4028;
   DATA[1745,14] := 1.0;
   DATA[1745,15] := 2.0;
   DATA[1745,16] := 1.0;
   DATA[1745,17] := 1.0;
   DATA[1745,18] := 1.0;
   DATA[1745,19] := 2.0;
   DATA[1745,20] := 148.808;
   DATA[1745,21] := 154.3707;
   DATA[1745,22] := 1.711595;
   DATA[1745,23] := 809.0618;
   DATA[1745,24] := 2.0;
   DATA[1745,25] := 2.0;
   DATA[1745,26] := 7.876058;
   DATA[1745,27] := 143.2966;
   DATA[1745,28] := 262.5288;
   DATA[1745,29] := 12.11228;
   DATA[1745,30] := 1.72302;
   DATA[1745,31] := 1.282183;
   DATA[1745,32] := 0.7352687;
   DATA[1745,33] := 0.3083624;
   DATA[1745,34] := 2.0;
   DATA[1745,35] := 250.0;
   DATA[1745,36] := 1.681991;
   DATA[1745,37] := 188.7977;
   DATA[1745,38] := 0.000128152;
   DATA[1745,39] := 1.0;
   DATA[1746,0] := 2.495916;
   DATA[1746,1] := 815.005;
   DATA[1746,2] := 2.0;
   DATA[1746,3] := 1.0;
   DATA[1746,4] := 262.625;
   DATA[1746,5] := 8.46501;
   DATA[1746,6] := 319.7385;
   DATA[1746,8] := 1.0;
   DATA[1746,9] := 1.0;
   DATA[1746,10] := 1.0;
   DATA[1746,11] := 19.73238;
   DATA[1746,12] := 2.210294;
   DATA[1746,13] := 835.0023;
   DATA[1746,14] := 1.0;
   DATA[1746,15] := 2.0;
   DATA[1746,16] := 1.0;
   DATA[1746,17] := 1.0;
   DATA[1746,18] := 1.0;
   DATA[1746,19] := 2.0;
   DATA[1746,20] := 148.808;
   DATA[1746,21] := 154.2938;
   DATA[1746,22] := 1.711595;
   DATA[1746,23] := 809.0233;
   DATA[1746,24] := 2.0;
   DATA[1746,25] := 2.0;
   DATA[1746,26] := 7.876058;
   DATA[1746,27] := 143.2966;
   DATA[1746,28] := 262.5288;
   DATA[1746,29] := 12.11228;
   DATA[1746,30] := 1.72302;
   DATA[1746,31] := 1.290893;
   DATA[1746,32] := 0.7352687;
   DATA[1746,33] := 0.3083624;
   DATA[1746,34] := 2.0;
   DATA[1746,35] := 250.0;
   DATA[1746,36] := 1.681991;
   DATA[1746,37] := 188.7977;
   DATA[1746,38] := 0.000128152;
   DATA[1746,39] := 1.0;
   DATA[1747,0] := 2.468693;
   DATA[1747,1] := 815.5153;
   DATA[1747,2] := 2.0;
   DATA[1747,3] := 1.0;
   DATA[1747,4] := 262.625;
   DATA[1747,5] := 8.46533;
   DATA[1747,6] := 319.7385;
   DATA[1747,8] := 1.0;
   DATA[1747,9] := 1.0;
   DATA[1747,10] := 1.0;
   DATA[1747,11] := 19.73238;
   DATA[1747,12] := 2.210294;
   DATA[1747,13] := 834.3614;
   DATA[1747,14] := 1.0;
   DATA[1747,15] := 2.0;
   DATA[1747,16] := 1.0;
   DATA[1747,17] := 1.0;
   DATA[1747,18] := 1.0;
   DATA[1747,19] := 2.0;
   DATA[1747,20] := 148.808;
   DATA[1747,21] := 154.2938;
   DATA[1747,22] := 1.711595;
   DATA[1747,23] := 808.8695;
   DATA[1747,24] := 2.0;
   DATA[1747,25] := 2.0;
   DATA[1747,26] := 7.876058;
   DATA[1747,27] := 143.2966;
   DATA[1747,28] := 262.5288;
   DATA[1747,29] := 12.11228;
   DATA[1747,30] := 1.72302;
   DATA[1747,31] := 1.286666;
   DATA[1747,32] := 0.7352687;
   DATA[1747,33] := 0.3083624;
   DATA[1747,34] := 2.0;
   DATA[1747,35] := 250.0;
   DATA[1747,36] := 1.681991;
   DATA[1747,37] := 188.7977;
   DATA[1747,38] := 0.000128152;
   DATA[1747,39] := 1.0;
   DATA[1748,0] := 2.459085;
   DATA[1748,1] := 815.7115;
   DATA[1748,2] := 2.0;
   DATA[1748,3] := 1.0;
   DATA[1748,4] := 262.625;
   DATA[1748,5] := 8.46533;
   DATA[1748,6] := 319.7385;
   DATA[1748,8] := 1.0;
   DATA[1748,9] := 1.0;
   DATA[1748,10] := 1.0;
   DATA[1748,11] := 19.73238;
   DATA[1748,12] := 2.210294;
   DATA[1748,13] := 833.8007;
   DATA[1748,14] := 1.0;
   DATA[1748,15] := 2.0;
   DATA[1748,16] := 1.0;
   DATA[1748,17] := 1.0;
   DATA[1748,18] := 1.0;
   DATA[1748,19] := 2.0;
   DATA[1748,20] := 148.808;
   DATA[1748,21] := 154.0118;
   DATA[1748,22] := 1.711595;
   DATA[1748,23] := 808.8695;
   DATA[1748,24] := 2.0;
   DATA[1748,25] := 2.0;
   DATA[1748,26] := 7.876058;
   DATA[1748,27] := 143.2966;
   DATA[1748,28] := 262.5288;
   DATA[1748,29] := 12.11228;
   DATA[1748,30] := 1.723404;
   DATA[1748,31] := 1.287691;
   DATA[1748,32] := 0.7377012;
   DATA[1748,33] := 0.3083624;
   DATA[1748,34] := 2.0;
   DATA[1748,35] := 249.8718;
   DATA[1748,36] := 1.681991;
   DATA[1748,37] := 188.7977;
   DATA[1748,38] := 0.000128152;
   DATA[1748,39] := 1.0;
   DATA[1749,0] := 2.444031;
   DATA[1749,1] := 815.4761;
   DATA[1749,2] := 2.0;
   DATA[1749,3] := 1.0;
   DATA[1749,4] := 262.625;
   DATA[1749,5] := 8.46533;
   DATA[1749,6] := 319.7385;
   DATA[1749,8] := 1.0;
   DATA[1749,9] := 1.0;
   DATA[1749,10] := 1.0;
   DATA[1749,11] := 19.76439;
   DATA[1749,12] := 2.210294;
   DATA[1749,13] := 833.4802;
   DATA[1749,14] := 1.0;
   DATA[1749,15] := 2.0;
   DATA[1749,16] := 1.0;
   DATA[1749,17] := 1.0;
   DATA[1749,18] := 1.0;
   DATA[1749,19] := 2.0;
   DATA[1749,20] := 148.808;
   DATA[1749,21] := 154.0118;
   DATA[1749,22] := 1.711595;
   DATA[1749,23] := 808.6388;
   DATA[1749,24] := 2.0;
   DATA[1749,25] := 2.0;
   DATA[1749,26] := 7.876058;
   DATA[1749,27] := 143.2966;
   DATA[1749,28] := 262.5288;
   DATA[1749,29] := 12.11228;
   DATA[1749,30] := 1.724301;
   DATA[1749,31] := 1.282567;
   DATA[1749,32] := 0.7377012;
   DATA[1749,33] := 0.31022;
   DATA[1749,34] := 2.0;
   DATA[1749,35] := 249.7437;
   DATA[1749,36] := 1.681991;
   DATA[1749,37] := 188.7977;
   DATA[1749,38] := 0.000128152;
   DATA[1749,39] := 1.0;
   DATA[1750,0] := 2.428979;
   DATA[1750,1] := 815.9471;
   DATA[1750,2] := 2.0;
   DATA[1750,3] := 1.0;
   DATA[1750,4] := 262.625;
   DATA[1750,5] := 8.46533;
   DATA[1750,6] := 319.7385;
   DATA[1750,8] := 1.0;
   DATA[1750,9] := 1.0;
   DATA[1750,10] := 1.0;
   DATA[1750,11] := 19.7964;
   DATA[1750,12] := 2.210294;
   DATA[1750,13] := 832.9996;
   DATA[1750,14] := 1.0;
   DATA[1750,15] := 2.0;
   DATA[1750,16] := 1.0;
   DATA[1750,17] := 1.0;
   DATA[1750,18] := 1.0;
   DATA[1750,19] := 2.0;
   DATA[1750,20] := 148.808;
   DATA[1750,21] := 154.0118;
   DATA[1750,22] := 1.711595;
   DATA[1750,23] := 809.0233;
   DATA[1750,24] := 2.0;
   DATA[1750,25] := 2.0;
   DATA[1750,26] := 7.876058;
   DATA[1750,27] := 143.2966;
   DATA[1750,28] := 262.5288;
   DATA[1750,29] := 12.11228;
   DATA[1750,30] := 1.724301;
   DATA[1750,31] := 1.293967;
   DATA[1750,32] := 0.7359089;
   DATA[1750,33] := 0.3094513;
   DATA[1750,34] := 2.0;
   DATA[1750,35] := 249.7437;
   DATA[1750,36] := 1.681991;
   DATA[1750,37] := 188.7977;
   DATA[1750,38] := 0.000128152;
   DATA[1750,39] := 1.0;
   DATA[1751,0] := 2.424174;
   DATA[1751,1] := 816.1041;
   DATA[1751,2] := 2.0;
   DATA[1751,3] := 1.0;
   DATA[1751,4] := 262.625;
   DATA[1751,5] := 8.46533;
   DATA[1751,6] := 319.7385;
   DATA[1751,8] := 1.0;
   DATA[1751,9] := 1.0;
   DATA[1751,10] := 1.0;
   DATA[1751,11] := 19.7964;
   DATA[1751,12] := 2.209269;
   DATA[1751,13] := 832.2786;
   DATA[1751,14] := 1.0;
   DATA[1751,15] := 2.0;
   DATA[1751,16] := 1.0;
   DATA[1751,17] := 1.0;
   DATA[1751,18] := 1.0;
   DATA[1751,19] := 2.0;
   DATA[1751,20] := 148.808;
   DATA[1751,21] := 154.0118;
   DATA[1751,22] := 1.711595;
   DATA[1751,23] := 808.9849;
   DATA[1751,24] := 2.0;
   DATA[1751,25] := 2.0;
   DATA[1751,26] := 7.876058;
   DATA[1751,27] := 143.2966;
   DATA[1751,28] := 262.5288;
   DATA[1751,29] := 12.11228;
   DATA[1751,30] := 1.725583;
   DATA[1751,31] := 1.301652;
   DATA[1751,32] := 0.7353967;
   DATA[1751,33] := 0.3086827;
   DATA[1751,34] := 2.0;
   DATA[1751,35] := 249.7437;
   DATA[1751,36] := 1.681991;
   DATA[1751,37] := 188.7977;
   DATA[1751,38] := 0.000128152;
   DATA[1751,39] := 1.0;
   DATA[1752,0] := 2.424174;
   DATA[1752,1] := 816.3788;
   DATA[1752,2] := 2.0;
   DATA[1752,3] := 1.0;
   DATA[1752,4] := 262.625;
   DATA[1752,5] := 8.46533;
   DATA[1752,6] := 319.7385;
   DATA[1752,8] := 1.0;
   DATA[1752,9] := 1.0;
   DATA[1752,10] := 1.0;
   DATA[1752,11] := 19.76439;
   DATA[1752,12] := 2.209269;
   DATA[1752,13] := 831.6778;
   DATA[1752,14] := 1.0;
   DATA[1752,15] := 2.0;
   DATA[1752,16] := 1.0;
   DATA[1752,17] := 1.0;
   DATA[1752,18] := 1.0;
   DATA[1752,19] := 2.0;
   DATA[1752,20] := 148.808;
   DATA[1752,21] := 154.1912;
   DATA[1752,22] := 1.711595;
   DATA[1752,23] := 809.254;
   DATA[1752,24] := 2.0;
   DATA[1752,25] := 2.0;
   DATA[1752,26] := 7.876058;
   DATA[1752,27] := 143.476;
   DATA[1752,28] := 262.5288;
   DATA[1752,29] := 12.11228;
   DATA[1752,30] := 1.725583;
   DATA[1752,31] := 1.29307;
   DATA[1752,32] := 0.7353967;
   DATA[1752,33] := 0.3081062;
   DATA[1752,34] := 2.0;
   DATA[1752,35] := 249.8398;
   DATA[1752,36] := 1.681991;
   DATA[1752,37] := 188.7977;
   DATA[1752,38] := 0.000128152;
   DATA[1752,39] := 1.0;
   DATA[1753,0] := 2.447234;
   DATA[1753,1] := 816.8499;
   DATA[1753,2] := 2.0;
   DATA[1753,3] := 1.0;
   DATA[1753,4] := 262.625;
   DATA[1753,5] := 8.46533;
   DATA[1753,6] := 319.7385;
   DATA[1753,8] := 1.0;
   DATA[1753,9] := 1.0;
   DATA[1753,10] := 1.0;
   DATA[1753,11] := 19.76439;
   DATA[1753,12] := 2.209269;
   DATA[1753,13] := 830.8367;
   DATA[1753,14] := 1.0;
   DATA[1753,15] := 2.0;
   DATA[1753,16] := 1.0;
   DATA[1753,17] := 1.0;
   DATA[1753,18] := 1.0;
   DATA[1753,19] := 2.0;
   DATA[1753,20] := 148.808;
   DATA[1753,21] := 154.1912;
   DATA[1753,22] := 1.711595;
   DATA[1753,23] := 809.0233;
   DATA[1753,24] := 2.0;
   DATA[1753,25] := 2.0;
   DATA[1753,26] := 7.876058;
   DATA[1753,27] := 143.476;
   DATA[1753,28] := 262.5288;
   DATA[1753,29] := 12.11228;
   DATA[1753,30] := 1.725583;
   DATA[1753,31] := 1.286025;
   DATA[1753,32] := 0.7353967;
   DATA[1753,33] := 0.3081062;
   DATA[1753,34] := 2.0;
   DATA[1753,35] := 249.8718;
   DATA[1753,36] := 1.681991;
   DATA[1753,37] := 188.7977;
   DATA[1753,38] := 0.000128152;
   DATA[1753,39] := 1.0;
   DATA[1754,0] := 2.493675;
   DATA[1754,1] := 817.6742;
   DATA[1754,2] := 2.0;
   DATA[1754,3] := 1.0;
   DATA[1754,4] := 262.625;
   DATA[1754,5] := 8.46533;
   DATA[1754,6] := 319.7385;
   DATA[1754,8] := 1.0;
   DATA[1754,9] := 1.0;
   DATA[1754,10] := 1.0;
   DATA[1754,11] := 19.76439;
   DATA[1754,12] := 2.209269;
   DATA[1754,13] := 830.5563;
   DATA[1754,14] := 1.0;
   DATA[1754,15] := 2.0;
   DATA[1754,16] := 1.0;
   DATA[1754,17] := 1.0;
   DATA[1754,18] := 1.0;
   DATA[1754,19] := 2.0;
   DATA[1754,20] := 148.808;
   DATA[1754,21] := 154.1912;
   DATA[1754,22] := 1.711595;
   DATA[1754,23] := 809.254;
   DATA[1754,24] := 2.0;
   DATA[1754,25] := 2.0;
   DATA[1754,26] := 7.876058;
   DATA[1754,27] := 143.476;
   DATA[1754,28] := 262.5288;
   DATA[1754,29] := 12.11228;
   DATA[1754,30] := 1.725327;
   DATA[1754,31] := 1.274881;
   DATA[1754,32] := 0.7353967;
   DATA[1754,33] := 0.3081062;
   DATA[1754,34] := 2.0;
   DATA[1754,35] := 249.8718;
   DATA[1754,36] := 1.681991;
   DATA[1754,37] := 188.7977;
   DATA[1754,38] := 0.000128152;
   DATA[1754,39] := 1.0;
   DATA[1754,40] := 1.0;
   DATA[1755,0] := 2.535951;
   DATA[1755,1] := 817.949;
   DATA[1755,2] := 2.0;
   DATA[1755,3] := 1.0;
   DATA[1755,4] := 262.625;
   DATA[1755,5] := 8.46533;
   DATA[1755,6] := 319.7385;
   DATA[1755,8] := 1.0;
   DATA[1755,9] := 1.0;
   DATA[1755,10] := 1.0;
   DATA[1755,11] := 19.76439;
   DATA[1755,12] := 2.209269;
   DATA[1755,13] := 829.5549;
   DATA[1755,14] := 1.0;
   DATA[1755,15] := 2.0;
   DATA[1755,16] := 1.0;
   DATA[1755,17] := 1.0;
   DATA[1755,18] := 1.0;
   DATA[1755,19] := 2.0;
   DATA[1755,20] := 148.808;
   DATA[1755,21] := 154.1912;
   DATA[1755,22] := 1.711595;
   DATA[1755,23] := 809.2156;
   DATA[1755,24] := 2.0;
   DATA[1755,25] := 2.0;
   DATA[1755,26] := 7.876058;
   DATA[1755,27] := 143.476;
   DATA[1755,28] := 262.4007;
   DATA[1755,29] := 12.11228;
   DATA[1755,30] := 1.725327;
   DATA[1755,31] := 1.280646;
   DATA[1755,32] := 0.7353967;
   DATA[1755,33] := 0.3081062;
   DATA[1755,34] := 2.0;
   DATA[1755,35] := 249.8718;
   DATA[1755,36] := 1.681991;
   DATA[1755,37] := 188.7977;
   DATA[1755,38] := 0.000128152;
   DATA[1755,39] := 1.0;
   DATA[1755,40] := 1.0;
   DATA[1756,0] := 2.535951;
   DATA[1756,1] := 817.949;
   DATA[1756,2] := 2.0;
   DATA[1756,3] := 1.0;
   DATA[1756,4] := 262.625;
   DATA[1756,5] := 8.46533;
   DATA[1756,6] := 319.7385;
   DATA[1756,8] := 1.0;
   DATA[1756,9] := 1.0;
   DATA[1756,10] := 1.0;
   DATA[1756,11] := 19.76439;
   DATA[1756,12] := 2.209269;
   DATA[1756,13] := 829.5549;
   DATA[1756,14] := 1.0;
   DATA[1756,15] := 2.0;
   DATA[1756,16] := 1.0;
   DATA[1756,17] := 1.0;
   DATA[1756,18] := 1.0;
   DATA[1756,19] := 2.0;
   DATA[1756,20] := 148.808;
   DATA[1756,21] := 154.1912;
   DATA[1756,22] := 1.711595;
   DATA[1756,23] := 809.2156;
   DATA[1756,24] := 2.0;
   DATA[1756,25] := 2.0;
   DATA[1756,26] := 7.876058;
   DATA[1756,27] := 143.476;
   DATA[1756,28] := 262.4007;
   DATA[1756,29] := 12.11228;
   DATA[1756,30] := 1.725327;
   DATA[1756,31] := 1.280646;
   DATA[1756,32] := 0.7353967;
   DATA[1756,33] := 0.3081062;
   DATA[1756,34] := 2.0;
   DATA[1756,35] := 249.8718;
   DATA[1756,36] := 1.681991;
   DATA[1756,37] := 188.7977;
   DATA[1756,38] := 0.000128152;
   DATA[1756,39] := 1.0;
   DATA[1756,40] := 1.0;
   DATA[1757,0] := 2.5699;
   DATA[1757,1] := 818.4592;
   DATA[1757,2] := 2.0;
   DATA[1757,3] := 1.0;
   DATA[1757,4] := 262.625;
   DATA[1757,5] := 8.46533;
   DATA[1757,6] := 319.7385;
   DATA[1757,8] := 1.0;
   DATA[1757,9] := 1.0;
   DATA[1757,10] := 1.0;
   DATA[1757,11] := 19.76439;
   DATA[1757,12] := 2.209269;
   DATA[1757,13] := 828.9942;
   DATA[1757,14] := 1.0;
   DATA[1757,15] := 2.0;
   DATA[1757,16] := 1.0;
   DATA[1757,17] := 1.0;
   DATA[1757,18] := 1.0;
   DATA[1757,19] := 2.0;
   DATA[1757,20] := 148.808;
   DATA[1757,21] := 154.1912;
   DATA[1757,22] := 1.711595;
   DATA[1757,23] := 809.0233;
   DATA[1757,24] := 2.0;
   DATA[1757,25] := 2.0;
   DATA[1757,26] := 7.876058;
   DATA[1757,27] := 143.476;
   DATA[1757,28] := 262.3366;
   DATA[1757,29] := 12.11228;
   DATA[1757,30] := 1.725327;
   DATA[1757,31] := 1.289996;
   DATA[1757,32] := 0.7353967;
   DATA[1757,33] := 0.3081062;
   DATA[1757,34] := 2.0;
   DATA[1757,35] := 249.8718;
   DATA[1757,36] := 1.681991;
   DATA[1757,37] := 188.7977;
   DATA[1757,38] := 0.000128152;
   DATA[1757,39] := 1.0;
   DATA[1757,40] := 1.0;
   DATA[1758,0] := 2.610575;
   DATA[1758,1] := 818.8911;
   DATA[1758,2] := 2.0;
   DATA[1758,3] := 1.0;
   DATA[1758,4] := 262.625;
   DATA[1758,5] := 8.46533;
   DATA[1758,6] := 319.7385;
   DATA[1758,8] := 1.0;
   DATA[1758,9] := 1.0;
   DATA[1758,10] := 1.0;
   DATA[1758,11] := 19.76439;
   DATA[1758,12] := 2.209269;
   DATA[1758,13] := 828.2732;
   DATA[1758,14] := 1.0;
   DATA[1758,15] := 2.0;
   DATA[1758,16] := 1.0;
   DATA[1758,17] := 1.0;
   DATA[1758,18] := 1.0;
   DATA[1758,19] := 2.0;
   DATA[1758,20] := 148.808;
   DATA[1758,21] := 154.1912;
   DATA[1758,22] := 1.711595;
   DATA[1758,23] := 808.9464;
   DATA[1758,24] := 2.0;
   DATA[1758,25] := 2.0;
   DATA[1758,26] := 7.876058;
   DATA[1758,27] := 143.476;
   DATA[1758,28] := 262.3366;
   DATA[1758,29] := 12.11228;
   DATA[1758,30] := 1.725327;
   DATA[1758,31] := 1.299603;
   DATA[1758,32] := 0.7353967;
   DATA[1758,33] := 0.3081062;
   DATA[1758,34] := 2.0;
   DATA[1758,35] := 250.0801;
   DATA[1758,36] := 1.681991;
   DATA[1758,37] := 188.974;
   DATA[1758,38] := 0.000128152;
   DATA[1758,39] := 1.0;
   DATA[1758,40] := 1.0;
   DATA[1759,0] := 2.635557;
   DATA[1759,1] := 818.6948;
   DATA[1759,2] := 2.0;
   DATA[1759,3] := 1.0;
   DATA[1759,4] := 262.625;
   DATA[1759,5] := 8.46533;
   DATA[1759,6] := 319.9436;
   DATA[1759,8] := 1.0;
   DATA[1759,9] := 1.0;
   DATA[1759,10] := 1.0;
   DATA[1759,11] := 19.76439;
   DATA[1759,12] := 2.209269;
   DATA[1759,13] := 827.9528;
   DATA[1759,14] := 1.0;
   DATA[1759,15] := 2.0;
   DATA[1759,16] := 1.0;
   DATA[1759,17] := 1.0;
   DATA[1759,18] := 1.0;
   DATA[1759,19] := 2.0;
   DATA[1759,20] := 148.808;
   DATA[1759,21] := 154.1912;
   DATA[1759,22] := 1.711595;
   DATA[1759,23] := 808.7926;
   DATA[1759,24] := 2.0;
   DATA[1759,25] := 2.0;
   DATA[1759,26] := 7.876058;
   DATA[1759,27] := 143.476;
   DATA[1759,28] := 262.3366;
   DATA[1759,29] := 12.11228;
   DATA[1759,30] := 1.725327;
   DATA[1759,31] := 1.301652;
   DATA[1759,32] := 0.7353967;
   DATA[1759,33] := 0.3086186;
   DATA[1759,34] := 2.0;
   DATA[1759,35] := 250.1923;
   DATA[1759,36] := 1.681991;
   DATA[1759,37] := 188.974;
   DATA[1759,38] := 0.000128152;
   DATA[1759,39] := 1.0;
   DATA[1759,40] := 1.0;
   DATA[1760,0] := 2.657336;
   DATA[1760,1] := 819.3228;
   DATA[1760,2] := 2.0;
   DATA[1760,3] := 1.0;
   DATA[1760,4] := 262.625;
   DATA[1760,5] := 8.46533;
   DATA[1760,6] := 319.9436;
   DATA[1760,8] := 1.0;
   DATA[1760,9] := 1.0;
   DATA[1760,10] := 1.0;
   DATA[1760,11] := 19.76439;
   DATA[1760,12] := 2.209269;
   DATA[1760,13] := 827.4321;
   DATA[1760,14] := 1.0;
   DATA[1760,15] := 2.0;
   DATA[1760,16] := 1.0;
   DATA[1760,17] := 1.0;
   DATA[1760,18] := 1.0;
   DATA[1760,19] := 2.0;
   DATA[1760,20] := 148.808;
   DATA[1760,21] := 154.1912;
   DATA[1760,22] := 1.711595;
   DATA[1760,23] := 808.9464;
   DATA[1760,24] := 2.0;
   DATA[1760,25] := 2.0;
   DATA[1760,26] := 7.876058;
   DATA[1760,27] := 143.476;
   DATA[1760,28] := 262.3366;
   DATA[1760,29] := 12.11228;
   DATA[1760,30] := 1.725327;
   DATA[1760,31] := 1.284745;
   DATA[1760,32] := 0.7353967;
   DATA[1760,33] := 0.3086186;
   DATA[1760,34] := 2.0;
   DATA[1760,35] := 250.1923;
   DATA[1760,36] := 1.681991;
   DATA[1760,37] := 188.974;
   DATA[1760,38] := 0.000128152;
   DATA[1760,39] := 1.0;
   DATA[1760,40] := 1.0;
   DATA[1761,0] := 2.663741;
   DATA[1761,1] := 819.7938;
   DATA[1761,2] := 2.0;
   DATA[1761,3] := 1.0;
   DATA[1761,4] := 262.625;
   DATA[1761,5] := 8.46533;
   DATA[1761,6] := 319.9436;
   DATA[1761,8] := 1.0;
   DATA[1761,9] := 1.0;
   DATA[1761,10] := 1.0;
   DATA[1761,11] := 19.72598;
   DATA[1761,12] := 2.209269;
   DATA[1761,13] := 826.8713;
   DATA[1761,14] := 1.0;
   DATA[1761,15] := 2.0;
   DATA[1761,16] := 1.0;
   DATA[1761,17] := 1.0;
   DATA[1761,18] := 1.0;
   DATA[1761,19] := 2.0;
   DATA[1761,20] := 148.808;
   DATA[1761,21] := 154.1912;
   DATA[1761,22] := 1.71262;
   DATA[1761,23] := 808.9464;
   DATA[1761,24] := 2.0;
   DATA[1761,25] := 2.0;
   DATA[1761,26] := 7.876058;
   DATA[1761,27] := 143.476;
   DATA[1761,28] := 262.3366;
   DATA[1761,29] := 12.11228;
   DATA[1761,30] := 1.725327;
   DATA[1761,31] := 1.273473;
   DATA[1761,32] := 0.7353967;
   DATA[1761,33] := 0.3086186;
   DATA[1761,34] := 2.0;
   DATA[1761,35] := 250.1923;
   DATA[1761,36] := 1.681991;
   DATA[1761,37] := 189.0541;
   DATA[1761,38] := 0.000128152;
   DATA[1761,39] := 1.0;
   DATA[1761,40] := 1.0;
   DATA[1762,0] := 2.641642;
   DATA[1762,1] := 820.0686;
   DATA[1762,2] := 2.0;
   DATA[1762,3] := 1.0;
   DATA[1762,4] := 262.625;
   DATA[1762,5] := 8.46533;
   DATA[1762,6] := 319.9436;
   DATA[1762,8] := 1.0;
   DATA[1762,9] := 1.0;
   DATA[1762,10] := 1.0;
   DATA[1762,11] := 19.70677;
   DATA[1762,12] := 2.210678;
   DATA[1762,13] := 826.3907;
   DATA[1762,14] := 1.0;
   DATA[1762,15] := 2.0;
   DATA[1762,16] := 1.0;
   DATA[1762,17] := 1.0;
   DATA[1762,18] := 1.0;
   DATA[1762,19] := 2.0;
   DATA[1762,20] := 148.808;
   DATA[1762,21] := 154.4219;
   DATA[1762,22] := 1.714029;
   DATA[1762,23] := 808.9849;
   DATA[1762,24] := 2.0;
   DATA[1762,25] := 2.0;
   DATA[1762,26] := 7.876058;
   DATA[1762,27] := 143.476;
   DATA[1762,28] := 262.3366;
   DATA[1762,29] := 12.11228;
   DATA[1762,30] := 1.726352;
   DATA[1762,31] := 1.26425;
   DATA[1762,32] := 0.7353967;
   DATA[1762,33] := 0.3086186;
   DATA[1762,34] := 2.0;
   DATA[1762,35] := 250.1923;
   DATA[1762,36] := 1.681991;
   DATA[1762,37] := 189.0541;
   DATA[1762,38] := 0.000128152;
   DATA[1762,39] := 1.0;
   DATA[1762,40] := 1.0;
   DATA[1763,0] := 2.629792;
   DATA[1763,1] := 820.4611;
   DATA[1763,2] := 2.0;
   DATA[1763,3] := 1.0;
   DATA[1763,4] := 262.625;
   DATA[1763,5] := 8.46533;
   DATA[1763,6] := 319.9436;
   DATA[1763,8] := 1.0;
   DATA[1763,9] := 1.0;
   DATA[1763,10] := 1.0;
   DATA[1763,11] := 19.70677;
   DATA[1763,12] := 2.210678;
   DATA[1763,13] := 826.2705;
   DATA[1763,14] := 1.0;
   DATA[1763,15] := 2.0;
   DATA[1763,16] := 1.0;
   DATA[1763,17] := 1.0;
   DATA[1763,18] := 1.0;
   DATA[1763,19] := 2.0;
   DATA[1763,20] := 148.808;
   DATA[1763,21] := 154.4219;
   DATA[1763,22] := 1.716464;
   DATA[1763,23] := 809.7155;
   DATA[1763,24] := 2.0;
   DATA[1763,25] := 2.0;
   DATA[1763,26] := 7.876058;
   DATA[1763,27] := 143.476;
   DATA[1763,28] := 262.3366;
   DATA[1763,29] := 12.11228;
   DATA[1763,30] := 1.727378;
   DATA[1763,31] := 1.262073;
   DATA[1763,32] := 0.7353967;
   DATA[1763,33] := 0.3086186;
   DATA[1763,34] := 2.0;
   DATA[1763,35] := 250.1923;
   DATA[1763,36] := 1.681991;
   DATA[1763,37] := 189.2143;
   DATA[1763,38] := 0.000128152;
   DATA[1763,39] := 1.0;
   DATA[1763,40] := 1.0;
   DATA[1764,0] := 2.621145;
   DATA[1764,1] := 821.2855;
   DATA[1764,2] := 2.0;
   DATA[1764,3] := 1.0;
   DATA[1764,4] := 262.625;
   DATA[1764,5] := 8.46533;
   DATA[1764,6] := 319.7898;
   DATA[1764,8] := 1.0;
   DATA[1764,9] := 1.0;
   DATA[1764,10] := 1.0;
   DATA[1764,11] := 19.70677;
   DATA[1764,12] := 2.210678;
   DATA[1764,13] := 825.6296;
   DATA[1764,14] := 1.0;
   DATA[1764,15] := 2.0;
   DATA[1764,16] := 1.0;
   DATA[1764,17] := 1.0;
   DATA[1764,18] := 1.0;
   DATA[1764,19] := 2.0;
   DATA[1764,20] := 148.808;
   DATA[1764,21] := 154.4219;
   DATA[1764,22] := 1.717105;
   DATA[1764,23] := 809.7924;
   DATA[1764,24] := 2.0;
   DATA[1764,25] := 2.0;
   DATA[1764,26] := 7.876058;
   DATA[1764,27] := 143.476;
   DATA[1764,28] := 262.3366;
   DATA[1764,29] := 12.11228;
   DATA[1764,30] := 1.727378;
   DATA[1764,31] := 1.270911;
   DATA[1764,32] := 0.7353967;
   DATA[1764,33] := 0.3086186;
   DATA[1764,34] := 2.0;
   DATA[1764,35] := 250.1923;
   DATA[1764,36] := 1.681991;
   DATA[1764,37] := 189.2143;
   DATA[1764,38] := 0.000128152;
   DATA[1764,39] := 1.0;
   DATA[1764,40] := 1.0;
   DATA[1765,0] := 2.612497;
   DATA[1765,1] := 821.2855;
   DATA[1765,2] := 2.0;
   DATA[1765,3] := 1.0;
   DATA[1765,4] := 262.625;
   DATA[1765,5] := 8.46533;
   DATA[1765,6] := 319.7898;
   DATA[1765,8] := 1.0;
   DATA[1765,9] := 1.0;
   DATA[1765,10] := 1.0;
   DATA[1765,11] := 19.65555;
   DATA[1765,12] := 2.210678;
   DATA[1765,13] := 824.9888;
   DATA[1765,14] := 1.0;
   DATA[1765,15] := 2.0;
   DATA[1765,16] := 1.0;
   DATA[1765,17] := 1.0;
   DATA[1765,18] := 1.0;
   DATA[1765,19] := 2.0;
   DATA[1765,20] := 148.808;
   DATA[1765,21] := 154.4219;
   DATA[1765,22] := 1.717105;
   DATA[1765,23] := 810.3307;
   DATA[1765,24] := 2.0;
   DATA[1765,25] := 2.0;
   DATA[1765,26] := 7.876058;
   DATA[1765,27] := 143.476;
   DATA[1765,28] := 262.3366;
   DATA[1765,29] := 12.11228;
   DATA[1765,30] := 1.727378;
   DATA[1765,31] := 1.271551;
   DATA[1765,32] := 0.7353967;
   DATA[1765,33] := 0.3086186;
   DATA[1765,34] := 2.0;
   DATA[1765,35] := 250.1923;
   DATA[1765,36] := 1.681991;
   DATA[1765,37] := 189.0861;
   DATA[1765,38] := 0.000128152;
   DATA[1765,39] := 1.0;
   DATA[1765,40] := 1.0;
   DATA[1766,0] := 2.601928;
   DATA[1766,1] := 821.4817;
   DATA[1766,2] := 2.0;
   DATA[1766,3] := 1.0;
   DATA[1766,4] := 262.625;
   DATA[1766,5] := 8.46533;
   DATA[1766,6] := 319.7898;
   DATA[1766,8] := 1.0;
   DATA[1766,9] := 1.0;
   DATA[1766,10] := 1.0;
   DATA[1766,11] := 19.63634;
   DATA[1766,12] := 2.209269;
   DATA[1766,13] := 824.5482;
   DATA[1766,14] := 1.0;
   DATA[1766,15] := 2.0;
   DATA[1766,16] := 1.0;
   DATA[1766,17] := 1.0;
   DATA[1766,18] := 1.0;
   DATA[1766,19] := 2.0;
   DATA[1766,20] := 148.808;
   DATA[1766,21] := 154.4219;
   DATA[1766,22] := 1.717105;
   DATA[1766,23] := 810.5614;
   DATA[1766,24] := 2.0;
   DATA[1766,25] := 2.0;
   DATA[1766,26] := 7.876058;
   DATA[1766,27] := 143.476;
   DATA[1766,28] := 262.3366;
   DATA[1766,29] := 12.11228;
   DATA[1766,30] := 1.727378;
   DATA[1766,31] := 1.280517;
   DATA[1766,32] := 0.7353967;
   DATA[1766,33] := 0.3080421;
   DATA[1766,34] := 2.0;
   DATA[1766,35] := 250.1923;
   DATA[1766,36] := 1.681991;
   DATA[1766,37] := 189.0861;
   DATA[1766,38] := 0.000128152;
   DATA[1766,39] := 1.0;
   DATA[1766,40] := 1.0;
   DATA[1767,0] := 2.585274;
   DATA[1767,1] := 821.8743;
   DATA[1767,2] := 2.0;
   DATA[1767,3] := 1.0;
   DATA[1767,4] := 262.625;
   DATA[1767,5] := 8.46533;
   DATA[1767,6] := 319.7898;
   DATA[1767,8] := 1.0;
   DATA[1767,9] := 1.0;
   DATA[1767,10] := 1.0;
   DATA[1767,11] := 19.63634;
   DATA[1767,12] := 2.208884;
   DATA[1767,13] := 823.9474;
   DATA[1767,14] := 1.0;
   DATA[1767,15] := 2.0;
   DATA[1767,16] := 1.0;
   DATA[1767,17] := 1.0;
   DATA[1767,18] := 1.0;
   DATA[1767,19] := 2.0;
   DATA[1767,20] := 148.808;
   DATA[1767,21] := 154.4219;
   DATA[1767,22] := 1.717105;
   DATA[1767,23] := 810.9459;
   DATA[1767,24] := 2.0;
   DATA[1767,25] := 2.0;
   DATA[1767,26] := 7.876058;
   DATA[1767,27] := 143.7067;
   DATA[1767,28] := 262.4007;
   DATA[1767,29] := 12.11228;
   DATA[1767,30] := 1.725711;
   DATA[1767,31] := 1.281927;
   DATA[1767,32] := 0.7353967;
   DATA[1767,33] := 0.3080421;
   DATA[1767,34] := 2.0;
   DATA[1767,35] := 250.1923;
   DATA[1767,36] := 1.681991;
   DATA[1767,37] := 188.974;
   DATA[1767,38] := 0.000128152;
   DATA[1767,39] := 1.0;
   DATA[1767,40] := 1.0;
   DATA[1768,0] := 2.566698;
   DATA[1768,1] := 822.2275;
   DATA[1768,2] := 2.0;
   DATA[1768,3] := 1.0;
   DATA[1768,4] := 262.625;
   DATA[1768,5] := 8.46533;
   DATA[1768,6] := 319.7898;
   DATA[1768,8] := 1.0;
   DATA[1768,9] := 1.0;
   DATA[1768,10] := 1.0;
   DATA[1768,11] := 19.63634;
   DATA[1768,12] := 2.208884;
   DATA[1768,13] := 823.5469;
   DATA[1768,14] := 1.0;
   DATA[1768,15] := 2.0;
   DATA[1768,16] := 1.0;
   DATA[1768,17] := 1.0;
   DATA[1768,18] := 1.0;
   DATA[1768,19] := 2.0;
   DATA[1768,20] := 148.808;
   DATA[1768,21] := 154.4219;
   DATA[1768,22] := 1.717105;
